C07311=1150.846,-117.168,-42.980,178.656,5.934,149.460
C07312=1150.851,-117.418,-42.971,178.654,5.933,149.460
C07313=1150.857,-117.668,-42.963,178.652,5.933,149.461
C07314=1150.862,-117.917,-42.954,178.650,5.933,149.461
C07315=1150.868,-118.167,-42.945,178.648,5.933,149.462
C07316=1150.873,-118.417,-42.936,178.646,5.932,149.462
C07317=1150.878,-118.667,-42.929,178.644,5.931,149.463
C07318=1150.883,-118.916,-42.920,178.642,5.931,149.463
C07319=1150.888,-119.166,-42.911,178.640,5.930,149.464
C07320=1150.894,-119.416,-42.903,178.638,5.931,149.464
C07321=1150.900,-119.666,-42.895,178.636,5.930,149.465
C07322=1150.905,-119.916,-42.886,178.634,5.930,149.465
C07323=1150.910,-120.165,-42.877,178.632,5.929,149.466
C07324=1150.915,-120.415,-42.868,178.630,5.929,149.466
C07325=1150.921,-120.665,-42.860,178.628,5.929,149.467
C07326=1150.926,-120.915,-42.851,178.627,5.929,149.467
C07327=1150.932,-121.165,-42.842,178.624,5.928,149.468
C07328=1150.937,-121.414,-42.834,178.622,5.928,149.469
C07329=1150.943,-121.664,-42.826,178.620,5.928,149.469
C07330=1150.948,-121.914,-42.817,178.619,5.928,149.470
C07331=1150.954,-122.163,-42.808,178.616,5.927,149.470
C07332=1150.959,-122.413,-42.801,178.615,5.927,149.471
C07333=1150.964,-122.663,-42.792,178.613,5.926,149.471
C07334=1150.969,-122.913,-42.783,178.611,5.926,149.472
C07335=1150.975,-123.163,-42.775,178.609,5.926,149.472
C07336=1150.980,-123.413,-42.766,178.606,5.925,149.473
C07337=1150.985,-123.663,-42.757,178.604,5.925,149.473
C07338=1150.991,-123.912,-42.749,178.602,5.924,149.474
C07339=1150.997,-124.162,-42.741,178.601,5.924,149.474
C07340=1151.001,-124.412,-42.733,178.598,5.924,149.475
C07341=1151.007,-124.662,-42.724,178.597,5.924,149.475
C07342=1151.012,-124.911,-42.716,178.595,5.923,149.476
C07343=1151.018,-125.162,-42.707,178.593,5.923,149.476
C07344=1151.023,-125.411,-42.699,178.591,5.922,149.477
C07345=1151.029,-125.661,-42.690,178.589,5.923,149.477
C07346=1151.034,-125.910,-42.683,178.587,5.922,149.478
C07347=1151.039,-126.160,-42.674,178.585,5.922,149.478
C07348=1151.045,-126.411,-42.666,178.583,5.921,149.479
C07349=1151.050,-126.660,-42.657,178.581,5.921,149.479
C07350=1151.056,-126.910,-42.649,178.579,5.921,149.480
C07351=1151.061,-127.160,-42.640,178.577,5.921,149.480
C07352=1151.066,-127.409,-42.632,178.575,5.920,149.481
C07353=1151.071,-127.659,-42.624,178.574,5.920,149.481
C07354=1151.077,-127.909,-42.615,178.571,5.919,149.482
C07355=1151.083,-128.159,-42.607,178.569,5.920,149.482
C07356=1150.661,-128.171,-42.650,178.566,5.922,149.484
C07357=1150.656,-127.920,-42.658,178.568,5.923,149.484
C07358=1150.651,-127.670,-42.667,178.570,5.923,149.483
C07359=1150.645,-127.420,-42.675,178.572,5.924,149.483
C07360=1150.640,-127.171,-42.683,178.574,5.924,149.482
C07361=1150.635,-126.922,-42.691,178.576,5.925,149.482
C07362=1150.629,-126.671,-42.700,178.577,5.925,149.481
C07363=1150.624,-126.421,-42.708,178.580,5.925,149.481
C07364=1150.618,-126.172,-42.716,178.581,5.925,149.480
C07365=1150.613,-125.922,-42.725,178.584,5.926,149.479
C07366=1150.608,-125.672,-42.733,178.585,5.926,149.479
C07367=1150.602,-125.423,-42.741,178.588,5.926,149.478
C07368=1150.597,-125.173,-42.750,178.589,5.926,149.478
C07369=1150.592,-124.922,-42.758,178.591,5.927,149.477
C07370=1150.586,-124.673,-42.767,178.593,5.927,149.477
C07371=1150.580,-124.423,-42.775,178.595,5.928,149.477
C07372=1150.576,-124.173,-42.783,178.597,5.928,149.476
C07373=1150.570,-123.924,-42.792,178.599,5.929,149.476
C07374=1150.565,-123.673,-42.800,178.601,5.928,149.475
C07375=1150.559,-123.424,-42.809,178.603,5.929,149.474
C07376=1150.554,-123.174,-42.818,178.605,5.929,149.474
C07377=1150.548,-122.924,-42.826,178.607,5.930,149.473
C07378=1150.543,-122.674,-42.835,178.609,5.929,149.473
C07379=1150.537,-122.425,-42.843,178.611,5.930,149.472
C07380=1150.533,-122.175,-42.851,178.612,5.930,149.472
C07381=1150.527,-121.925,-42.860,178.615,5.931,149.471
C07382=1150.522,-121.676,-42.868,178.617,5.932,149.471
C07383=1150.516,-121.425,-42.876,178.619,5.931,149.470
C07384=1150.511,-121.175,-42.885,178.621,5.932,149.470
C07385=1150.505,-120.926,-42.894,178.623,5.932,149.469
C07386=1150.500,-120.676,-42.902,178.625,5.933,149.469
C07387=1150.495,-120.426,-42.911,178.627,5.933,149.468
C07388=1150.489,-120.176,-42.920,178.629,5.933,149.468
C07389=1150.484,-119.927,-42.928,178.630,5.933,149.467
C07390=1150.478,-119.677,-42.936,178.633,5.934,149.467
C07391=1150.473,-119.427,-42.945,178.635,5.934,149.466
C07392=1150.467,-119.178,-42.954,178.637,5.934,149.466
C07393=1150.462,-118.928,-42.963,178.638,5.934,149.465
C07394=1150.457,-118.678,-42.970,178.641,5.935,149.465
C07395=1150.452,-118.428,-42.979,178.642,5.935,149.464
C07396=1150.446,-118.179,-42.988,178.644,5.936,149.464
C07397=1150.441,-117.929,-42.997,178.646,5.936,149.463
C07398=1150.436,-117.678,-43.005,178.649,5.936,149.462
C07399=1150.430,-117.429,-43.013,178.651,5.937,149.462
C07400=1150.425,-117.179,-43.022,178.652,5.937,149.461
C07401=1150.420,-116.929,-43.031,178.655,5.938,149.461
C07402=1150.415,-116.680,-43.040,178.656,5.938,149.460
C07403=1150.409,-116.430,-43.049,178.658,5.938,149.460
C07404=1150.403,-116.180,-43.057,178.660,5.938,149.460
C07405=1150.398,-115.930,-43.066,178.663,5.939,149.459
C07406=1150.393,-115.680,-43.075,178.664,5.939,149.458
C07407=1150.387,-115.431,-43.083,178.666,5.939,149.458
C07408=1150.382,-115.181,-43.092,178.668,5.939,149.457
C07409=1150.377,-114.931,-43.101,178.670,5.940,149.457
C07410=1150.371,-114.681,-43.110,178.672,5.941,149.456
C07411=1150.365,-114.431,-43.119,178.674,5.941,149.456
C07412=1150.360,-114.182,-43.127,178.677,5.941,149.455
C07413=1150.355,-113.932,-43.136,178.678,5.941,149.455
C07414=1150.349,-113.682,-43.145,178.681,5.942,149.454
C07415=1150.344,-113.432,-43.154,178.682,5.942,149.454
C07416=1150.338,-113.183,-43.162,178.684,5.943,149.453
C07417=1150.333,-112.933,-43.171,178.686,5.943,149.453
C07418=1150.328,-112.683,-43.180,178.689,5.943,149.452
C07419=1150.323,-112.433,-43.188,178.691,5.944,149.452
C07420=1150.317,-112.183,-43.197,178.692,5.944,149.451
C07421=1150.312,-111.934,-43.206,178.695,5.944,149.451
C07422=1150.307,-111.684,-43.215,178.696,5.944,149.450
C07423=1150.301,-111.434,-43.224,178.698,5.945,149.450
C07424=1150.295,-111.184,-43.233,178.700,5.945,149.449
C07425=1150.290,-110.934,-43.242,178.703,5.945,149.448
C07426=1150.285,-110.684,-43.251,178.705,5.946,149.448
C07427=1150.279,-110.435,-43.259,178.706,5.946,149.447
C07428=1150.274,-110.185,-43.268,178.709,5.947,149.447
C07429=1150.269,-109.935,-43.277,178.711,5.947,149.446
C07430=1150.264,-109.685,-43.286,178.713,5.947,149.446
C07431=1150.259,-109.436,-43.295,178.715,5.947,149.445
C07432=1150.254,-109.186,-43.304,178.717,5.948,149.445
C07433=1150.247,-108.936,-43.313,178.719,5.949,149.444
C07434=1150.242,-108.686,-43.322,178.721,5.949,149.444
C07435=1150.237,-108.437,-43.331,178.723,5.949,149.443
C07436=1150.232,-108.187,-43.340,178.725,5.949,149.443
C07437=1150.226,-107.937,-43.349,178.727,5.950,149.442
C07438=1150.221,-107.687,-43.358,178.729,5.950,149.442
C07439=1150.215,-107.437,-43.367,178.731,5.951,149.441
C07440=1150.210,-107.188,-43.376,178.733,5.951,149.440
C07441=1150.204,-106.938,-43.384,178.735,5.951,149.440
C07442=1150.199,-106.688,-43.393,178.737,5.952,149.439
C07443=1150.194,-106.438,-43.402,178.739,5.952,149.439
C07444=1150.189,-106.188,-43.411,178.741,5.952,149.438
C07445=1150.183,-105.939,-43.421,178.744,5.953,149.438
C07446=1150.178,-105.689,-43.430,178.745,5.953,149.437
C07447=1150.173,-105.439,-43.439,178.748,5.953,149.437
C07448=1150.168,-105.189,-43.448,178.749,5.953,149.436
C07449=1150.162,-104.940,-43.457,178.751,5.954,149.436
C07450=1150.156,-104.690,-43.466,178.753,5.954,149.435
C07451=1150.151,-104.440,-43.475,178.756,5.954,149.435
C07452=1150.146,-104.190,-43.484,178.758,5.955,149.434
C07453=1150.141,-103.941,-43.493,178.759,5.955,149.434
C07454=1150.135,-103.691,-43.503,178.762,5.956,149.433
C07455=1150.130,-103.441,-43.512,178.764,5.956,149.432
C07456=1150.125,-103.191,-43.521,178.766,5.956,149.432
C07457=1150.119,-102.919,-43.531,178.768,5.957,149.431
C07458=1150.113,-102.647,-43.540,178.771,5.957,149.431
C07459=1150.107,-102.375,-43.550,178.772,5.957,149.430
C07460=1150.101,-102.103,-43.560,178.775,5.958,149.430
C07461=1150.096,-101.853,-43.570,178.777,5.959,149.429
C07462=1150.091,-101.603,-43.579,178.779,5.958,149.429
C07463=1150.086,-101.354,-43.588,178.781,5.959,149.428
C07464=1150.080,-101.103,-43.597,178.784,5.960,149.427
C07465=1150.074,-100.854,-43.606,178.785,5.960,149.427
C07466=1150.070,-100.604,-43.616,178.787,5.960,149.426
C07467=1150.064,-100.354,-43.625,178.789,5.960,149.426
C07468=1150.059,-100.104,-43.634,178.791,5.961,149.425
C07469=1150.053,-99.854,-43.643,178.794,5.961,149.425
C07470=1150.049,-99.605,-43.653,178.795,5.961,149.424
C07471=1150.043,-99.355,-43.662,178.798,5.962,149.424
C07472=1150.037,-99.105,-43.671,178.799,5.962,149.423
C07473=1150.032,-98.855,-43.680,178.802,5.962,149.423
C07474=1150.027,-98.606,-43.690,178.804,5.963,149.422
C07475=1150.022,-98.356,-43.699,178.806,5.963,149.422
C07476=1150.016,-98.106,-43.709,178.808,5.964,149.421
C07477=1150.011,-97.857,-43.718,178.811,5.964,149.420
C07478=1150.006,-97.607,-43.727,178.812,5.964,149.420
C07479=1150.000,-97.357,-43.737,178.814,5.965,149.419
C07480=1149.995,-97.107,-43.746,178.816,5.965,149.419
C07481=1149.990,-96.857,-43.755,178.819,5.965,149.418
C07482=1149.984,-96.607,-43.765,178.821,5.966,149.418
C07483=1149.979,-96.358,-43.774,178.822,5.966,149.417
C07484=1149.974,-96.108,-43.783,178.825,5.967,149.417
C07485=1149.968,-95.858,-43.793,178.827,5.967,149.416
C07486=1149.963,-95.609,-43.802,178.829,5.967,149.416
C07487=1149.957,-95.359,-43.812,178.831,5.968,149.415
C07488=1149.952,-95.109,-43.821,178.833,5.968,149.415
C07489=1149.946,-94.859,-43.831,178.835,5.968,149.414
C07490=1149.941,-94.609,-43.840,178.838,5.969,149.413
C07491=1149.936,-94.360,-43.849,178.839,5.969,149.413
C07492=1149.930,-94.110,-43.859,178.841,5.970,149.412
C07493=1149.925,-93.860,-43.868,178.844,5.970,149.412
C07494=1149.920,-93.611,-43.878,178.846,5.970,149.411
C07495=1149.914,-93.361,-43.887,178.848,5.971,149.411
C07496=1149.909,-93.111,-43.897,178.850,5.972,149.410
C07497=1149.904,-92.861,-43.906,178.852,5.971,149.410
C07498=1149.898,-92.612,-43.915,178.854,5.972,149.409
C07499=1149.893,-92.362,-43.925,178.857,5.973,149.409
C07500=1149.888,-92.112,-43.934,178.858,5.973,149.408
C07501=1149.882,-91.863,-43.944,178.861,5.973,149.407
C07502=1149.877,-91.613,-43.953,178.863,5.974,149.407
C07503=1149.871,-91.363,-43.963,178.865,5.974,149.406
C07504=1149.867,-91.113,-43.973,178.867,5.975,149.406
C07505=1149.861,-90.863,-43.983,178.869,5.975,149.405
C07506=1149.856,-90.613,-43.992,178.871,5.975,149.405
C07507=1149.850,-90.364,-44.002,178.873,5.976,149.404
C07508=1149.845,-90.114,-44.011,178.875,5.975,149.404
C07509=1149.840,-89.864,-44.021,178.877,5.976,149.403
C07510=1149.834,-89.614,-44.030,178.880,5.977,149.403
C07511=1149.829,-89.365,-44.040,178.881,5.977,149.402
C07512=1149.824,-89.115,-44.049,178.884,5.977,149.401
C07513=1149.818,-88.866,-44.059,178.886,5.978,149.401
C07514=1149.814,-88.615,-44.068,178.888,5.978,149.400
C07515=1149.808,-88.365,-44.079,178.890,5.979,149.400
C07516=1149.803,-88.116,-44.088,178.893,5.979,149.399
C07517=1149.797,-87.866,-44.098,178.894,5.979,149.399
C07518=1149.792,-87.617,-44.107,178.896,5.980,149.398
C07519=1149.786,-87.367,-44.117,178.899,5.980,149.398
C07520=1149.781,-87.117,-44.127,178.901,5.981,149.397
C07521=1149.776,-86.867,-44.136,178.903,5.981,149.397
C07522=1149.771,-86.617,-44.147,178.905,5.982,149.396
C07523=1149.766,-86.368,-44.156,178.908,5.982,149.395
C07524=1149.760,-86.118,-44.166,178.909,5.982,149.395
C07525=1149.755,-85.868,-44.175,178.912,5.983,149.394
C07526=1149.749,-85.618,-44.185,178.914,5.983,149.394
C07527=1149.744,-85.369,-44.195,178.916,5.983,149.393
C07528=1149.739,-85.119,-44.205,178.918,5.984,149.393
C07529=1149.733,-84.869,-44.214,178.920,5.985,149.392
C07530=1149.729,-84.619,-44.224,178.922,5.984,149.392
C07531=1149.723,-84.370,-44.234,178.924,5.985,149.391
C07532=1149.717,-84.120,-44.244,178.927,5.986,149.391
C07533=1149.712,-83.870,-44.253,178.929,5.985,149.390
C07534=1149.707,-83.620,-44.264,178.931,5.986,149.389
C07535=1149.702,-83.370,-44.273,178.933,5.987,149.389
C07536=1149.696,-83.121,-44.283,178.935,5.987,149.388
C07537=1149.691,-82.871,-44.293,178.937,5.987,149.388
C07538=1149.686,-82.622,-44.303,178.940,5.988,149.387
C07539=1149.681,-82.371,-44.313,178.942,5.989,149.387
C07540=1149.675,-82.122,-44.323,178.944,5.988,149.386
C07541=1149.670,-81.872,-44.333,178.946,5.989,149.386
C07542=1149.665,-81.623,-44.343,178.948,5.990,149.385
C07543=1149.659,-81.373,-44.352,178.950,5.990,149.384
C07544=1149.654,-81.123,-44.362,178.952,5.990,149.384
C07545=1149.649,-80.873,-44.372,178.955,5.991,149.383
C07546=1149.643,-80.624,-44.383,178.957,5.991,149.383
C07547=1149.638,-80.374,-44.392,178.959,5.991,149.382
C07548=1149.633,-80.124,-44.402,178.961,5.992,149.382
C07549=1149.627,-79.874,-44.412,178.964,5.993,149.381
C07550=1149.622,-79.624,-44.423,178.965,5.993,149.381
C07551=1149.617,-79.375,-44.431,178.968,5.993,149.380
C07552=1149.611,-79.125,-44.442,178.970,5.994,149.379
C07553=1149.606,-78.875,-44.452,178.972,5.994,149.379
C07554=1149.601,-78.626,-44.462,178.974,5.994,149.378
C07555=1149.596,-78.376,-44.472,178.976,5.995,149.378
C07556=1149.590,-78.127,-44.482,178.979,5.996,149.377
C07557=1149.585,-77.876,-44.492,178.980,5.996,149.377
C07558=1149.580,-77.626,-44.502,178.983,5.996,149.376
C07559=1149.574,-77.377,-44.512,178.985,5.997,149.376
C07560=1149.569,-77.127,-44.522,178.988,5.997,149.375
C07561=1149.563,-76.856,-44.533,178.990,5.997,149.374
C07562=1149.558,-76.584,-44.545,178.992,5.998,149.374
C07563=1149.552,-76.312,-44.555,178.994,5.998,149.373
C07564=1149.546,-76.042,-44.566,178.997,5.999,149.373
C07565=1149.540,-75.792,-44.576,178.999,6.000,149.372
C07566=1149.536,-75.542,-44.586,179.001,5.999,149.371
C07567=1149.530,-75.293,-44.596,179.003,6.000,149.371
C07568=1149.524,-75.043,-44.607,179.005,6.001,149.370
C07569=1149.519,-74.793,-44.617,179.008,6.001,149.370
C07570=1149.514,-74.543,-44.627,179.010,6.001,149.369
C07571=1149.508,-74.294,-44.638,179.012,6.002,149.369
C07572=1149.504,-74.044,-44.648,179.014,6.002,149.368
C07573=1149.498,-73.794,-44.658,179.017,6.003,149.368
C07574=1149.493,-73.545,-44.668,179.018,6.003,149.367
C07575=1149.487,-73.295,-44.678,179.021,6.004,149.366
C07576=1149.482,-73.044,-44.688,179.023,6.004,149.366
C07577=1149.476,-72.795,-44.698,179.025,6.005,149.365
C07578=1149.471,-72.545,-44.708,179.027,6.005,149.365
C07579=1149.466,-72.295,-44.719,179.030,6.005,149.364
C07580=1149.461,-72.046,-44.729,179.032,6.006,149.364
C07581=1149.455,-71.796,-44.739,179.034,6.007,149.363
C07582=1149.451,-71.547,-44.750,179.036,6.007,149.363
C07583=1149.445,-71.297,-44.760,179.039,6.007,149.362
C07584=1149.439,-71.047,-44.771,179.041,6.008,149.361
C07585=1149.434,-70.797,-44.781,179.043,6.008,149.361
C07586=1149.429,-70.548,-44.791,179.045,6.008,149.360
C07587=1149.425,-70.298,-44.801,179.047,6.009,149.360
C07588=1149.419,-70.048,-44.812,179.050,6.010,149.359
C07589=1149.413,-69.799,-44.822,179.052,6.010,149.359
C07590=1149.408,-69.548,-44.832,179.054,6.010,149.358
C07591=1149.403,-69.299,-44.843,179.056,6.011,149.358
C07592=1149.397,-69.049,-44.853,179.059,6.011,149.357
C07593=1149.392,-68.799,-44.863,179.061,6.012,149.356
C07594=1149.387,-68.550,-44.874,179.062,6.012,149.356
C07595=1149.382,-68.299,-44.884,179.065,6.012,149.355
C07596=1149.376,-68.050,-44.895,179.067,6.013,149.355
C07597=1149.371,-67.801,-44.905,179.069,6.014,149.354
C07598=1149.366,-67.551,-44.916,179.072,6.014,149.354
C07599=1149.360,-67.301,-44.926,179.074,6.014,149.353
C07600=1149.355,-67.051,-44.937,179.076,6.015,149.353
C07601=1149.349,-66.801,-44.947,179.079,6.015,149.352
C07602=1149.344,-66.552,-44.957,179.081,6.016,149.351
C07603=1149.339,-66.302,-44.968,179.083,6.016,149.351
C07604=1149.334,-66.053,-44.979,179.085,6.017,149.350
C07605=1149.329,-65.802,-44.989,179.087,6.017,149.350
C07606=1149.323,-65.553,-44.999,179.090,6.018,149.349
C07607=1149.318,-65.302,-45.010,179.092,6.018,149.349
C07608=1149.313,-65.054,-45.021,179.094,6.018,149.348
C07609=1149.307,-64.804,-45.031,179.096,6.019,149.347
C07610=1149.302,-64.554,-45.042,179.099,6.020,149.347
C07611=1149.297,-64.304,-45.052,179.101,6.020,149.346
C07612=1149.292,-64.055,-45.063,179.103,6.021,149.346
C07613=1149.286,-63.805,-45.073,179.105,6.021,149.345
C07614=1149.281,-63.555,-45.084,179.107,6.022,149.345
C07615=1149.276,-63.305,-45.094,179.110,6.022,149.344
C07616=1149.271,-63.056,-45.105,179.112,6.023,149.344
C07617=1149.265,-62.806,-45.116,179.114,6.022,149.343
C07618=1149.260,-62.556,-45.126,179.116,6.023,149.342
C07619=1149.255,-62.306,-45.136,179.119,6.024,149.342
C07620=1149.250,-62.057,-45.148,179.121,6.024,149.341
C07621=1149.244,-61.807,-45.158,179.123,6.025,149.341
C07622=1149.239,-61.558,-45.168,179.125,6.025,149.340
C07623=1149.234,-61.308,-45.179,179.128,6.025,149.340
C07624=1149.229,-61.058,-45.190,179.130,6.026,149.339
C07625=1149.224,-60.808,-45.200,179.132,6.027,149.338
C07626=1149.218,-60.559,-45.212,179.135,6.027,149.338
C07627=1149.213,-60.309,-45.222,179.137,6.028,149.337
C07628=1149.208,-60.058,-45.233,179.139,6.028,149.337
C07629=1149.202,-59.810,-45.244,179.141,6.029,149.336
C07630=1149.197,-59.559,-45.254,179.143,6.029,149.336
C07631=1149.192,-59.310,-45.265,179.146,6.030,149.335
C07632=1149.187,-59.060,-45.276,179.148,6.030,149.335
C07633=1149.181,-58.811,-45.286,179.150,6.030,149.334
C07634=1149.177,-58.561,-45.297,179.152,6.031,149.333
C07635=1149.170,-58.311,-45.308,179.155,6.032,149.333
C07636=1149.166,-58.061,-45.319,179.157,6.032,149.332
C07637=1149.160,-57.812,-45.330,179.159,6.033,149.332
C07638=1149.155,-57.562,-45.340,179.162,6.034,149.331
C07639=1149.150,-57.313,-45.351,179.164,6.033,149.331
C07640=1149.145,-57.063,-45.362,179.166,6.034,149.330
C07641=1149.139,-56.813,-45.374,179.169,6.034,149.329
C07642=1149.134,-56.563,-45.384,179.171,6.035,149.329
C07643=1149.129,-56.313,-45.395,179.173,6.036,149.328
C07644=1149.123,-56.064,-45.405,179.176,6.036,149.328
C07645=1149.119,-55.814,-45.417,179.177,6.036,149.327
C07646=1149.113,-55.565,-45.427,179.180,6.037,149.326
C07647=1149.108,-55.315,-45.439,179.182,6.037,149.326
C07648=1149.103,-55.065,-45.449,179.184,6.038,149.326
C07649=1149.097,-54.816,-45.460,179.187,6.039,149.325
C07650=1149.092,-54.565,-45.471,179.189,6.039,149.324
C07651=1149.086,-54.316,-45.482,179.191,6.039,149.324
C07652=1149.081,-54.066,-45.493,179.193,6.040,149.323
C07653=1149.077,-53.816,-45.504,179.196,6.041,149.323
C07654=1149.071,-53.567,-45.514,179.198,6.041,149.322
C07655=1149.066,-53.317,-45.526,179.200,6.042,149.321
C07656=1149.060,-53.067,-45.536,179.203,6.043,149.321
C07657=1149.055,-52.818,-45.548,179.205,6.042,149.320
C07658=1149.051,-52.568,-45.559,179.207,6.043,149.320
C07659=1149.044,-52.318,-45.570,179.210,6.043,149.319
C07660=1149.040,-52.068,-45.581,179.212,6.044,149.319
C07661=1149.034,-51.819,-45.591,179.214,6.045,149.318
C07662=1149.029,-51.569,-45.603,179.217,6.045,149.317
C07663=1149.024,-51.319,-45.615,179.219,6.046,149.317
C07664=1149.018,-51.070,-45.625,179.221,6.046,149.316
C07665=1149.013,-50.799,-45.637,179.223,6.046,149.316
C07666=1149.007,-50.528,-45.649,179.226,6.047,149.315
C07667=1149.002,-50.258,-45.661,179.228,6.048,149.315
C07668=1148.996,-49.987,-45.673,179.231,6.049,149.314
C07669=1148.991,-49.737,-45.685,179.233,6.049,149.313
C07670=1148.985,-49.488,-45.696,179.235,6.049,149.313
C07671=1148.980,-49.238,-45.706,179.238,6.050,149.312
C07672=1148.975,-48.988,-45.718,179.240,6.050,149.312
C07673=1148.970,-48.739,-45.729,179.242,6.051,149.311
C07674=1148.965,-48.489,-45.740,179.245,6.052,149.311
C07675=1148.959,-48.239,-45.751,179.247,6.052,149.310
C07676=1148.954,-47.990,-45.762,179.249,6.052,149.309
C07677=1148.948,-47.740,-45.774,179.252,6.053,149.309
C07678=1148.943,-47.490,-45.785,179.254,6.054,149.308
C07679=1148.938,-47.241,-45.796,179.256,6.054,149.308
C07680=1148.933,-46.991,-45.808,179.259,6.055,149.307
C07681=1148.928,-46.741,-45.819,179.261,6.056,149.307
C07682=1148.922,-46.491,-45.830,179.263,6.056,149.306
C07683=1148.917,-46.242,-45.841,179.266,6.057,149.305
C07684=1148.912,-45.992,-45.852,179.268,6.057,149.305
C07685=1148.907,-45.742,-45.864,179.270,6.057,149.304
C07686=1148.901,-45.493,-45.874,179.272,6.058,149.304
C07687=1148.896,-45.243,-45.886,179.275,6.058,149.303
C07688=1148.891,-44.993,-45.898,179.277,6.059,149.303
C07689=1148.885,-44.744,-45.909,179.280,6.059,149.302
C07690=1148.880,-44.494,-45.920,179.282,6.060,149.301
C07691=1148.875,-44.244,-45.931,179.284,6.061,149.301
C07692=1148.870,-43.994,-45.943,179.287,6.061,149.300
C07693=1148.865,-43.745,-45.954,179.289,6.062,149.300
C07694=1148.859,-43.495,-45.966,179.291,6.062,149.299
C07695=1148.855,-43.246,-45.977,179.293,6.063,149.299
C07696=1148.849,-42.996,-45.989,179.295,6.063,149.298
C07697=1148.844,-42.747,-46.000,179.298,6.064,149.297
C07698=1148.838,-42.497,-46.012,179.300,6.065,149.297
C07699=1148.833,-42.246,-46.022,179.303,6.065,149.296
C07700=1148.828,-41.997,-46.034,179.305,6.066,149.296
C07701=1148.823,-41.747,-46.045,179.307,6.067,149.295
C07702=1148.817,-41.498,-46.057,179.310,6.067,149.295
C07703=1148.813,-41.248,-46.068,179.312,6.068,149.294
C07704=1148.807,-40.998,-46.080,179.315,6.068,149.293
C07705=1148.802,-40.749,-46.091,179.317,6.069,149.293
C07706=1148.796,-40.499,-46.103,179.319,6.069,149.292
C07707=1148.792,-40.250,-46.114,179.321,6.069,149.292
C07708=1148.786,-40.000,-46.126,179.323,6.070,149.291
C07709=1148.781,-39.750,-46.138,179.326,6.071,149.291
C07710=1148.776,-39.500,-46.149,179.328,6.071,149.290
C07711=1148.770,-39.251,-46.161,179.331,6.072,149.289
C07712=1148.765,-39.001,-46.172,179.333,6.073,149.289
C07713=1148.760,-38.751,-46.184,179.335,6.073,149.288
C07714=1148.755,-38.502,-46.195,179.338,6.074,149.288
C07715=1148.750,-38.252,-46.207,179.340,6.075,149.287
C07716=1148.744,-38.002,-46.219,179.343,6.075,149.287
C07717=1148.739,-37.753,-46.230,179.345,6.076,149.286
C07718=1148.734,-37.503,-46.242,179.348,6.076,149.285
C07719=1148.729,-37.253,-46.253,179.349,6.076,149.285
C07720=1148.724,-37.003,-46.265,179.351,6.077,149.284
C07721=1148.718,-36.753,-46.277,179.354,6.077,149.284
C07722=1148.714,-36.504,-46.288,179.356,6.078,149.283
C07723=1148.707,-36.255,-46.300,179.359,6.079,149.283
C07724=1148.702,-36.005,-46.312,179.361,6.079,149.282
C07725=1148.697,-35.755,-46.323,179.364,6.080,149.281
C07726=1148.692,-35.505,-46.335,179.366,6.081,149.281
C07727=1148.688,-35.256,-46.347,179.368,6.081,149.280
C07728=1148.682,-35.006,-46.359,179.371,6.082,149.280
C07729=1148.677,-34.756,-46.370,179.373,6.083,149.279
C07730=1148.672,-34.507,-46.382,179.376,6.083,149.279
C07731=1148.666,-34.257,-46.393,179.378,6.084,149.278
C07732=1148.661,-34.007,-46.405,179.380,6.084,149.277
C07733=1148.655,-33.758,-46.417,179.383,6.085,149.277
C07734=1148.651,-33.509,-46.429,179.385,6.086,149.276
C07735=1148.645,-33.259,-46.441,179.387,6.086,149.276
C07736=1148.640,-33.009,-46.453,179.390,6.087,149.275
C07737=1148.635,-32.759,-46.464,179.392,6.087,149.275
C07738=1148.630,-32.509,-46.476,179.395,6.088,149.274
C07739=1148.624,-32.259,-46.488,179.397,6.089,149.273
C07740=1148.620,-32.010,-46.500,179.399,6.089,149.273
C07741=1148.614,-31.761,-46.511,179.401,6.089,149.272
C07742=1148.608,-31.511,-46.523,179.404,6.090,149.272
C07743=1148.603,-31.261,-46.535,179.406,6.091,149.271
C07744=1148.599,-31.012,-46.547,179.408,6.091,149.271
C07745=1148.593,-30.762,-46.559,179.411,6.092,149.270
C07746=1148.588,-30.512,-46.571,179.413,6.092,149.269
C07747=1148.582,-30.262,-46.583,179.415,6.093,149.269
C07748=1148.578,-30.013,-46.595,179.418,6.094,149.268
C07749=1148.573,-29.763,-46.607,179.420,6.094,149.268
C07750=1148.567,-29.513,-46.619,179.422,6.095,149.267
C07751=1148.562,-29.264,-46.631,179.425,6.095,149.267
C07752=1148.557,-29.014,-46.643,179.427,6.096,149.266
C07753=1148.552,-28.764,-46.654,179.430,6.097,149.265
C07754=1148.546,-28.515,-46.666,179.432,6.097,149.265
C07755=1148.541,-28.265,-46.679,179.434,6.098,149.264
C07756=1148.536,-28.015,-46.691,179.437,6.099,149.264
C07757=1148.530,-27.765,-46.703,179.439,6.099,149.263
C07758=1148.526,-27.516,-46.715,179.442,6.100,149.263
C07759=1148.521,-27.266,-46.727,179.444,6.101,149.262
C07760=1148.516,-27.017,-46.739,179.447,6.101,149.261
C07761=1148.510,-26.767,-46.751,179.449,6.102,149.261
C07762=1148.505,-26.517,-46.763,179.452,6.102,149.260
C07763=1148.500,-26.268,-46.776,179.454,6.103,149.260
C07764=1148.495,-26.018,-46.787,179.456,6.104,149.259
C07765=1148.490,-25.769,-46.799,179.459,6.104,149.259
C07766=1148.484,-25.519,-46.811,179.461,6.105,149.258
C07767=1148.479,-25.269,-46.823,179.463,6.105,149.257
C07768=1148.474,-25.020,-46.836,179.466,6.106,149.257
C07769=1148.468,-24.749,-46.849,179.468,6.107,149.256
C07770=1148.463,-24.480,-46.861,179.470,6.107,149.256
C07771=1148.457,-24.210,-46.876,179.474,6.109,149.255
C07772=1148.451,-23.939,-46.889,179.476,6.109,149.254
C07773=1148.446,-23.689,-46.900,179.479,6.110,149.254
C07774=1148.441,-23.440,-46.913,179.481,6.110,149.253
C07775=1148.435,-23.190,-46.925,179.483,6.111,149.253
C07776=1148.430,-22.941,-46.938,179.486,6.112,149.252
C07777=1148.425,-22.691,-46.949,179.488,6.112,149.252
C07778=1148.421,-22.442,-46.961,179.490,6.113,149.251
C07779=1148.415,-22.192,-46.973,179.493,6.114,149.250
C07780=1148.410,-21.943,-46.986,179.495,6.114,149.250
C07781=1148.405,-21.693,-46.999,179.498,6.115,149.249
C07782=1148.399,-21.443,-47.010,179.500,6.116,149.249
C07783=1148.394,-21.194,-47.023,179.503,6.116,149.248
C07784=1148.389,-20.944,-47.035,179.505,6.117,149.248
C07785=1148.384,-20.695,-47.048,179.507,6.118,149.247
C07786=1148.378,-20.445,-47.059,179.510,6.118,149.246
C07787=1148.374,-20.195,-47.072,179.512,6.119,149.246
C07788=1148.369,-19.946,-47.085,179.515,6.119,149.245
C07789=1148.363,-19.696,-47.097,179.517,6.120,149.245
C07790=1148.358,-19.446,-47.109,179.520,6.120,149.244
C07791=1148.353,-19.196,-47.121,179.522,6.121,149.244
C07792=1148.348,-18.947,-47.134,179.524,6.122,149.243
C07793=1148.342,-18.698,-47.147,179.527,6.122,149.243
C07794=1148.337,-18.448,-47.158,179.529,6.123,149.242
C07795=1148.333,-18.198,-47.171,179.532,6.124,149.241
C07796=1148.327,-17.948,-47.185,179.534,6.125,149.241
C07797=1148.321,-17.698,-47.196,179.537,6.126,149.240
C07798=1148.316,-17.449,-47.209,179.539,6.126,149.240
C07799=1148.311,-17.200,-47.222,179.542,6.127,149.239
C07800=1148.306,-16.950,-47.234,179.544,6.128,149.239
C07801=1148.300,-16.700,-47.246,179.546,6.128,149.238
C07802=1148.296,-16.450,-47.259,179.549,6.129,149.237
C07803=1148.290,-16.200,-47.271,179.551,6.130,149.237
C07804=1148.285,-15.951,-47.284,179.554,6.130,149.236
C07805=1148.280,-15.702,-47.296,179.556,6.131,149.236
C07806=1148.275,-15.452,-47.309,179.558,6.131,149.235
C07807=1148.270,-15.202,-47.321,179.561,6.132,149.235
C07808=1148.264,-14.952,-47.334,179.563,6.133,149.234
C07809=1148.259,-14.703,-47.347,179.565,6.133,149.233
C07810=1148.254,-14.453,-47.359,179.568,6.134,149.233
C07811=1148.249,-14.204,-47.372,179.570,6.135,149.232
C07812=1148.244,-13.954,-47.384,179.573,6.136,149.232
C07813=1148.239,-13.704,-47.397,179.576,6.137,149.231
C07814=1148.234,-13.455,-47.410,179.578,6.137,149.231
C07815=1148.228,-13.205,-47.423,179.580,6.138,149.230
C07816=1148.223,-12.956,-47.435,179.583,6.139,149.229
C07817=1148.218,-12.706,-47.447,179.585,6.139,149.229
C07818=1148.213,-12.456,-47.460,179.587,6.140,149.228
C07819=1148.208,-12.207,-47.473,179.590,6.140,149.228
C07820=1148.203,-11.957,-47.485,179.592,6.141,149.227
C07821=1148.197,-11.708,-47.499,179.595,6.142,149.226
C07822=1148.192,-11.458,-47.512,179.597,6.142,149.226
C07823=1148.187,-11.208,-47.524,179.599,6.143,149.226
C07824=1148.182,-10.959,-47.537,179.603,6.144,149.225
C07825=1148.177,-10.709,-47.549,179.605,6.145,149.224
C07826=1148.171,-10.459,-47.562,179.607,6.146,149.224
C07827=1148.166,-10.209,-47.575,179.610,6.146,149.223
C07828=1148.161,-9.960,-47.587,179.612,6.147,149.223
C07829=1148.156,-9.711,-47.600,179.614,6.148,149.222
C07830=1148.151,-9.461,-47.614,179.617,6.148,149.221
C07831=1148.146,-9.211,-47.626,179.619,6.149,149.221
C07832=1148.141,-8.962,-47.639,179.621,6.150,149.220
C07833=1148.136,-8.712,-47.652,179.624,6.150,149.220
C07834=1148.130,-8.462,-47.665,179.627,6.152,149.219
C07835=1148.125,-8.213,-47.678,179.630,6.152,149.219
C07836=1148.120,-7.964,-47.690,179.632,6.153,149.218
C07837=1148.115,-7.714,-47.703,179.634,6.153,149.217
C07838=1148.110,-7.464,-47.716,179.637,6.154,149.217
C07839=1148.104,-7.215,-47.729,179.639,6.155,149.216
C07840=1148.100,-6.965,-47.742,179.641,6.155,149.216
C07841=1148.094,-6.715,-47.755,179.644,6.156,149.215
C07842=1148.089,-6.466,-47.768,179.646,6.157,149.215
C07843=1148.084,-6.216,-47.781,179.649,6.158,149.214
C07844=1148.079,-5.966,-47.794,179.652,6.159,149.213
C07845=1148.073,-5.717,-47.806,179.654,6.160,149.213
C07846=1148.069,-5.467,-47.819,179.657,6.160,149.212
C07847=1148.063,-5.218,-47.833,179.659,6.161,149.212
C07848=1148.058,-4.968,-47.846,179.661,6.161,149.211
C07849=1148.054,-4.718,-47.859,179.664,6.162,149.211
C07850=1148.048,-4.469,-47.872,179.666,6.162,149.210
C07851=1148.043,-4.219,-47.885,179.669,6.164,149.210
C07852=1148.038,-3.969,-47.898,179.671,6.165,149.209
C07853=1148.032,-3.720,-47.911,179.674,6.165,149.208
C07854=1148.027,-3.470,-47.923,179.676,6.166,149.208
C07855=1148.022,-3.221,-47.938,179.679,6.167,149.207
C07856=1148.017,-2.971,-47.950,179.681,6.167,149.207
C07857=1148.013,-2.721,-47.963,179.683,6.168,149.206
C07858=1148.007,-2.472,-47.976,179.686,6.169,149.206
C07859=1148.002,-2.222,-47.989,179.689,6.170,149.205
C07860=1147.996,-1.972,-48.003,179.691,6.171,149.204
C07861=1147.992,-1.723,-48.016,179.693,6.171,149.204
C07862=1147.987,-1.473,-48.029,179.696,6.172,149.203
C07863=1147.981,-1.224,-48.042,179.698,6.173,149.203
C07864=1147.976,-0.974,-48.055,179.701,6.173,149.202
C07865=1147.971,-0.725,-48.069,179.703,6.175,149.202
C07866=1147.966,-0.475,-48.082,179.706,6.175,149.201
C07867=1147.961,-0.225,-48.095,179.708,6.176,149.201
C07868=1147.956,0.024,-48.108,179.711,6.176,149.200
C07869=1147.950,0.273,-48.122,179.713,6.177,149.199
C07870=1147.945,0.523,-48.135,179.716,6.178,149.199
C07871=1147.940,0.773,-48.148,179.719,6.179,149.198
C07872=1147.935,1.023,-48.161,179.721,6.180,149.198
C07873=1147.929,1.292,-48.175,179.723,6.181,149.197
C07874=1147.923,1.562,-48.190,179.726,6.181,149.196
C07875=1147.919,1.831,-48.204,179.729,6.183,149.196
C07876=1147.913,2.101,-48.218,179.731,6.183,149.195
C07877=1147.907,2.350,-48.232,179.734,6.184,149.195
C07878=1147.903,2.600,-48.245,179.736,6.184,149.194
C07879=1147.897,2.849,-48.259,179.739,6.186,149.194
C07880=1147.892,3.098,-48.272,179.742,6.186,149.193
C07881=1147.887,3.348,-48.285,179.744,6.187,149.192
C07882=1147.882,3.597,-48.299,179.747,6.188,149.192
C07883=1147.877,3.848,-48.312,179.749,6.188,149.191
C07884=1147.872,4.096,-48.325,179.752,6.190,149.191
C07885=1147.867,4.347,-48.339,179.754,6.190,149.190
C07886=1147.861,4.596,-48.352,179.756,6.191,149.190
C07887=1147.857,4.846,-48.366,179.759,6.192,149.189
C07888=1147.851,5.095,-48.379,179.761,6.193,149.189
C07889=1147.847,5.345,-48.393,179.764,6.193,149.188
C07890=1147.841,5.594,-48.406,179.767,6.195,149.187
C07891=1147.836,5.844,-48.420,179.769,6.195,149.187
C07892=1147.831,6.094,-48.433,179.771,6.196,149.186
C07893=1147.826,6.343,-48.447,179.774,6.196,149.186
C07894=1147.821,6.593,-48.460,179.776,6.197,149.185
C07895=1147.816,6.842,-48.474,179.779,6.199,149.185
C07896=1147.810,7.092,-48.488,179.782,6.199,149.184
C07897=1147.806,7.341,-48.501,179.784,6.200,149.183
C07898=1147.800,7.591,-48.514,179.787,6.200,149.183
C07899=1147.795,7.840,-48.528,179.789,6.202,149.182
C07900=1147.790,8.090,-48.541,179.792,6.202,149.182
C07901=1147.785,8.339,-48.555,179.794,6.203,149.181
C07902=1147.779,8.590,-48.569,179.797,6.204,149.181
C07903=1147.775,8.839,-48.583,179.799,6.205,149.180
C07904=1147.769,9.089,-48.596,179.802,6.206,149.180
C07905=1147.764,9.338,-48.610,179.804,6.207,149.179
C07906=1147.759,9.587,-48.624,179.807,6.207,149.178
C07907=1147.754,9.837,-48.637,179.809,6.208,149.178
C07908=1147.749,10.086,-48.651,179.811,6.209,149.177
C07909=1147.744,10.336,-48.665,179.815,6.210,149.177
C07910=1147.739,10.586,-48.678,179.817,6.211,149.176
C07911=1147.734,10.835,-48.692,179.819,6.211,149.175
C07912=1147.728,11.086,-48.705,179.822,6.212,149.175
C07913=1147.723,11.335,-48.719,179.824,6.214,149.175
C07914=1147.719,11.584,-48.733,179.827,6.214,149.174
C07915=1147.713,11.834,-48.747,179.829,6.215,149.173
C07916=1147.708,12.083,-48.761,179.832,6.215,149.173
C07917=1147.703,12.333,-48.775,179.835,6.217,149.172
C07918=1147.698,12.583,-48.789,179.837,6.217,149.172
C07919=1147.693,12.832,-48.802,179.839,6.218,149.171
C07920=1147.688,13.082,-48.816,179.842,6.219,149.170
C07921=1147.682,13.331,-48.830,179.844,6.219,149.170
C07922=1147.677,13.581,-48.843,179.847,6.221,149.170
C07923=1147.672,13.831,-48.858,179.850,6.222,149.169
C07924=1147.667,14.079,-48.871,179.852,6.222,149.168
C07925=1147.662,14.329,-48.885,179.854,6.223,149.168
C07926=1147.657,14.580,-48.899,179.857,6.224,149.167
C07927=1147.651,14.829,-48.913,179.860,6.225,149.167
C07928=1147.646,15.078,-48.927,179.862,6.226,149.166
C07929=1147.642,15.328,-48.941,179.865,6.227,149.165
C07930=1147.637,15.577,-48.955,179.868,6.228,149.165
C07931=1147.631,15.827,-48.968,179.870,6.229,149.164
C07932=1147.627,16.077,-48.983,179.872,6.229,149.164
C07933=1147.622,16.326,-48.997,179.875,6.231,149.163
C07934=1147.616,16.575,-49.011,179.878,6.231,149.163
C07935=1147.611,16.825,-49.025,179.880,6.232,149.162
C07936=1147.606,17.075,-49.039,179.883,6.232,149.162
C07937=1147.601,17.324,-49.053,179.885,6.234,149.161
C07938=1147.596,17.574,-49.066,179.887,6.235,149.161
C07939=1147.591,17.824,-49.080,179.890,6.235,149.160
C07940=1147.585,18.073,-49.094,179.892,6.236,149.159
C07941=1147.581,18.322,-49.109,179.896,6.237,149.159
C07942=1147.576,18.572,-49.123,179.898,6.238,149.158
C07943=1147.571,18.822,-49.137,179.900,6.239,149.158
C07944=1147.565,19.071,-49.151,179.903,6.240,149.157
C07945=1147.560,19.320,-49.165,179.906,6.241,149.156
C07946=1147.555,19.570,-49.180,179.908,6.242,149.156
C07947=1147.550,19.820,-49.194,179.910,6.242,149.156
C07948=1147.545,20.069,-49.208,179.913,6.244,149.155
C07949=1147.540,20.319,-49.222,179.916,6.244,149.154
C07950=1147.535,20.568,-49.236,179.918,6.245,149.154
C07951=1147.530,20.818,-49.251,179.921,6.246,149.153
C07952=1147.524,21.067,-49.265,179.924,6.247,149.153
C07953=1147.519,21.317,-49.279,179.926,6.248,149.152
C07954=1147.514,21.566,-49.293,179.928,6.249,149.152
C07955=1147.509,21.816,-49.307,179.931,6.250,149.151
C07956=1147.504,22.066,-49.322,179.933,6.251,149.151
C07957=1147.499,22.315,-49.336,179.936,6.251,149.150
C07958=1147.494,22.565,-49.350,179.939,6.253,149.149
C07959=1147.489,22.814,-49.364,179.941,6.253,149.149
C07960=1147.484,23.064,-49.378,179.944,6.254,149.148
C07961=1147.479,23.314,-49.393,179.946,6.256,149.148
C07962=1147.473,23.563,-49.407,179.949,6.256,149.147
C07963=1147.469,23.812,-49.421,179.951,6.257,149.147
C07964=1147.464,24.062,-49.435,179.954,6.258,149.146
C07965=1147.459,24.311,-49.450,179.957,6.259,149.146
C07966=1147.454,24.561,-49.464,179.959,6.259,149.145
C07967=1147.449,24.811,-49.479,179.961,6.260,149.144
C07968=1147.443,25.060,-49.493,179.964,6.262,149.144
C07969=1147.438,25.310,-49.507,179.967,6.262,149.143
C07970=1147.433,25.559,-49.522,179.969,6.263,149.143
C07971=1147.428,25.808,-49.537,179.972,6.264,149.142
C07972=1147.423,26.058,-49.551,179.974,6.265,149.142
C07973=1147.418,26.308,-49.565,179.977,6.266,149.141
C07974=1147.413,26.557,-49.579,179.980,6.267,149.141
C07975=1147.408,26.807,-49.593,179.982,6.268,149.140
C07976=1147.403,27.056,-49.608,179.985,6.269,149.139
C07977=1147.397,27.325,-49.624,179.987,6.270,149.139
C07978=1147.392,27.594,-49.640,179.990,6.271,149.138
C07979=1147.387,27.863,-49.655,179.993,6.272,149.138
C07980=1147.381,28.132,-49.672,179.995,6.273,149.137
C07981=1147.376,28.382,-49.686,179.999,6.274,149.137
C07982=1147.371,28.632,-49.700,-179.999,6.275,149.136
C07983=1147.366,28.881,-49.715,-179.996,6.276,149.135
C07984=1147.361,29.130,-49.729,-179.994,6.277,149.135
C07985=1147.356,29.379,-49.744,-179.992,6.278,149.134
C07986=1147.350,29.629,-49.758,-179.988,6.279,149.134
C07987=1147.345,29.878,-49.773,-179.986,6.280,149.133
C07988=1147.340,30.128,-49.788,-179.984,6.280,149.133
C07989=1147.335,30.378,-49.802,-179.981,6.282,149.132
C07990=1147.330,30.627,-49.818,-179.978,6.282,149.132
C07991=1147.325,30.877,-49.832,-179.976,6.283,149.131
C07992=1147.320,31.127,-49.846,-179.973,6.285,149.131
C07993=1147.316,31.376,-49.861,-179.971,6.285,149.130
C07994=1147.310,31.626,-49.876,-179.968,6.286,149.130
C07995=1147.305,31.875,-49.891,-179.965,6.287,149.129
C07996=1147.300,32.125,-49.905,-179.963,6.288,149.128
C07997=1147.295,32.374,-49.919,-179.960,6.290,149.128
C07998=1147.290,32.624,-49.935,-179.958,6.290,149.127
C07999=1147.285,32.873,-49.949,-179.955,6.291,149.127
C08000=1147.280,33.123,-49.964,-179.952,6.293,149.126
C08001=1147.275,33.373,-49.979,-179.950,6.293,149.126
C08002=1147.270,33.622,-49.994,-179.947,6.294,149.125
C08003=1147.264,33.871,-50.008,-179.945,6.295,149.125
C08004=1147.259,34.120,-50.024,-179.942,6.296,149.124
C08005=1147.254,34.370,-50.038,-179.939,6.298,149.123
C08006=1147.249,34.619,-50.053,-179.937,6.298,149.123
C08007=1147.244,34.869,-50.068,-179.934,6.299,149.122
C08008=1147.240,35.119,-50.083,-179.932,6.300,149.122
C08009=1147.235,35.368,-50.097,-179.929,6.301,149.121
C08010=1147.229,35.618,-50.113,-179.927,6.302,149.121
C08011=1147.224,35.868,-50.127,-179.924,6.303,149.120
C08012=1147.220,36.117,-50.142,-179.921,6.304,149.120
C08013=1147.214,36.367,-50.157,-179.919,6.306,149.119
C08014=1147.209,36.616,-50.172,-179.916,6.306,149.119
C08015=1147.204,36.866,-50.187,-179.914,6.307,149.118
C08016=1147.199,37.115,-50.202,-179.911,6.308,149.118
C08017=1147.194,37.364,-50.217,-179.908,6.309,149.117
C08018=1147.189,37.614,-50.232,-179.906,6.311,149.116
C08019=1147.184,37.863,-50.247,-179.904,6.311,149.116
C08020=1147.179,38.112,-50.263,-179.900,6.313,149.115
C08021=1147.174,38.362,-50.277,-179.898,6.313,149.115
C08022=1147.168,38.612,-50.292,-179.895,6.314,149.114
C08023=1147.163,38.861,-50.307,-179.893,6.316,149.114
C08024=1147.158,39.111,-50.322,-179.890,6.316,149.113
C08025=1147.153,39.360,-50.337,-179.887,6.318,149.113
C08026=1147.148,39.609,-50.353,-179.885,6.319,149.112
C08027=1147.143,39.859,-50.367,-179.883,6.319,149.111
C08028=1147.138,40.109,-50.383,-179.880,6.321,149.111
C08029=1147.134,40.358,-50.398,-179.877,6.321,149.110
C08030=1147.128,40.608,-50.413,-179.874,6.323,149.110
C08031=1147.123,40.857,-50.428,-179.872,6.324,149.109
C08032=1147.118,41.107,-50.444,-179.869,6.325,149.109
C08033=1147.113,41.356,-50.459,-179.867,6.326,149.108
C08034=1147.107,41.606,-50.473,-179.864,6.326,149.108
C08035=1147.103,41.855,-50.488,-179.861,6.328,149.107
C08036=1147.097,42.104,-50.504,-179.859,6.329,149.107
C08037=1147.093,42.354,-50.519,-179.856,6.330,149.106
C08038=1147.088,42.604,-50.534,-179.854,6.331,149.106
C08039=1147.083,42.853,-50.549,-179.851,6.332,149.105
C08040=1147.078,43.102,-50.565,-179.848,6.333,149.105
C08041=1147.073,43.352,-50.580,-179.846,6.334,149.104
C08042=1147.068,43.601,-50.595,-179.843,6.335,149.103
C08043=1147.063,43.851,-50.611,-179.841,6.336,149.103
C08044=1147.058,44.101,-50.626,-179.838,6.337,149.103
C08045=1147.053,44.350,-50.641,-179.835,6.338,149.102
C08046=1147.048,44.599,-50.656,-179.833,6.340,149.101
C08047=1147.042,44.849,-50.672,-179.830,6.340,149.101
C08048=1147.037,45.098,-50.687,-179.827,6.342,149.100
C08049=1147.033,45.348,-50.703,-179.825,6.343,149.100
C08050=1147.028,45.597,-50.718,-179.822,6.344,149.099
C08051=1147.023,45.846,-50.733,-179.820,6.345,149.099
C08052=1147.018,46.096,-50.749,-179.817,6.345,149.098
C08053=1147.012,46.345,-50.764,-179.814,6.347,149.098
C08054=1147.008,46.595,-50.780,-179.812,6.348,149.097
C08055=1147.003,46.844,-50.795,-179.809,6.349,149.097
C08056=1146.997,47.094,-50.811,-179.807,6.350,149.096
C08057=1146.992,47.343,-50.825,-179.804,6.351,149.096
C08058=1146.988,47.594,-50.841,-179.801,6.352,149.095
C08059=1146.982,47.843,-50.857,-179.799,6.353,149.095
C08060=1146.978,48.092,-50.872,-179.796,6.354,149.094
C08061=1146.973,48.341,-50.888,-179.793,6.356,149.093
C08062=1146.968,48.591,-50.904,-179.791,6.356,149.093
C08063=1146.962,48.840,-50.920,-179.788,6.358,149.092
C08064=1146.958,49.089,-50.935,-179.786,6.359,149.092
C08065=1146.952,49.339,-50.950,-179.782,6.360,149.091
C08066=1146.948,49.589,-50.966,-179.780,6.361,149.091
C08067=1146.943,49.838,-50.981,-179.778,6.362,149.090
C08068=1146.938,50.087,-50.997,-179.775,6.363,149.090
C08069=1146.932,50.337,-51.012,-179.772,6.364,149.089
C08070=1146.927,50.587,-51.028,-179.770,6.365,149.089
C08071=1146.923,50.836,-51.043,-179.767,6.367,149.088
C08072=1146.917,51.085,-51.059,-179.765,6.367,149.088
C08073=1146.913,51.335,-51.076,-179.761,6.369,149.087
C08074=1146.907,51.584,-51.091,-179.759,6.370,149.087
C08075=1146.902,51.834,-51.107,-179.756,6.371,149.086
C08076=1146.897,52.083,-51.122,-179.754,6.372,149.085
C08077=1146.893,52.333,-51.138,-179.751,6.373,149.085
C08078=1146.887,52.582,-51.153,-179.749,6.374,149.085
C08079=1146.882,52.831,-51.170,-179.746,6.375,149.084
C08080=1146.877,53.081,-51.186,-179.744,6.376,149.083
C08081=1146.872,53.350,-51.203,-179.740,6.378,149.083
C08082=1146.867,53.618,-51.219,-179.738,6.379,149.082
C08083=1146.861,53.886,-51.236,-179.735,6.380,149.082
C08084=1146.856,54.155,-51.253,-179.732,6.381,149.081
C08085=1146.851,54.405,-51.269,-179.730,6.382,149.081
C08086=1146.846,54.654,-51.285,-179.727,6.383,149.080
C08087=1146.841,54.904,-51.300,-179.724,6.385,149.080
C08088=1146.836,55.153,-51.317,-179.721,6.386,149.079
C08089=1146.830,55.403,-51.332,-179.719,6.387,149.079
C08090=1146.826,55.653,-51.348,-179.716,6.388,149.078
C08091=1146.820,55.902,-51.364,-179.713,6.389,149.077
C08092=1146.816,56.151,-51.380,-179.711,6.390,149.077
C08093=1146.811,56.401,-51.396,-179.708,6.391,149.076
C08094=1146.806,56.650,-51.411,-179.706,6.392,149.076
C08095=1146.801,56.900,-51.428,-179.703,6.394,149.075
C08096=1146.796,57.149,-51.443,-179.700,6.394,149.075
C08097=1146.791,57.398,-51.460,-179.698,6.396,149.074
C08098=1146.786,57.648,-51.476,-179.695,6.397,149.074
C08099=1146.781,57.897,-51.491,-179.692,6.398,149.073
C08100=1146.776,58.147,-51.508,-179.690,6.399,149.073
C08101=1146.771,58.396,-51.524,-179.687,6.401,149.072
C08102=1146.766,58.645,-51.540,-179.684,6.402,149.072
C08103=1146.761,58.895,-51.556,-179.682,6.403,149.071
C08104=1146.756,59.144,-51.571,-179.679,6.404,149.071
C08105=1146.751,59.394,-51.588,-179.676,6.405,149.070
C08106=1146.746,59.643,-51.604,-179.674,6.407,149.070
C08107=1146.741,59.893,-51.620,-179.671,6.407,149.069
C08108=1146.736,60.142,-51.636,-179.668,6.409,149.069
C08109=1146.731,60.392,-51.653,-179.666,6.410,149.068
C08110=1146.726,60.641,-51.668,-179.663,6.411,149.068
C08111=1146.721,60.890,-51.684,-179.660,6.413,149.067
C08112=1146.716,61.140,-51.700,-179.658,6.413,149.067
C08113=1146.711,61.389,-51.717,-179.655,6.415,149.066
C08114=1146.706,61.639,-51.733,-179.653,6.416,149.066
C08115=1146.701,61.888,-51.749,-179.650,6.417,149.065
C08116=1146.696,62.138,-51.765,-179.647,6.418,149.064
C08117=1146.691,62.387,-51.781,-179.645,6.419,149.064
C08118=1146.686,62.636,-51.798,-179.642,6.421,149.064
C08119=1146.681,62.886,-51.814,-179.639,6.422,149.063
C08120=1146.676,63.135,-51.831,-179.636,6.423,149.062
C08121=1146.671,63.385,-51.846,-179.634,6.424,149.062
C08122=1146.666,63.634,-51.863,-179.631,6.425,149.061
C08123=1146.661,63.883,-51.879,-179.628,6.427,149.061
C08124=1146.656,64.133,-51.895,-179.626,6.428,149.060
C08125=1146.651,64.382,-51.912,-179.623,6.429,149.060
C08126=1146.647,64.632,-51.928,-179.621,6.430,149.059
C08127=1146.641,64.882,-51.945,-179.618,6.432,149.059
C08128=1146.636,65.130,-51.961,-179.615,6.433,149.058
C08129=1146.632,65.380,-51.978,-179.613,6.434,149.058
C08130=1146.626,65.629,-51.993,-179.610,6.435,149.057
C08131=1146.622,65.879,-52.010,-179.607,6.436,149.057
C08132=1146.617,66.128,-52.026,-179.605,6.438,149.056
C08133=1146.611,66.378,-52.043,-179.602,6.439,149.056
C08134=1146.606,66.627,-52.059,-179.599,6.440,149.055
C08135=1146.602,66.876,-52.076,-179.596,6.441,149.055
C08136=1146.597,67.126,-52.093,-179.594,6.442,149.054
C08137=1146.592,67.375,-52.108,-179.591,6.444,149.054
C08138=1146.587,67.625,-52.125,-179.588,6.445,149.053
C08139=1146.582,67.874,-52.142,-179.586,6.446,149.053
C08140=1146.577,68.123,-52.158,-179.583,6.447,149.052
C08141=1146.573,68.373,-52.175,-179.581,6.448,149.052
C08142=1146.566,68.622,-52.191,-179.578,6.450,149.051
C08143=1146.562,68.872,-52.208,-179.575,6.451,149.051
C08144=1146.557,69.121,-52.224,-179.573,6.452,149.050
C08145=1146.552,69.370,-52.241,-179.570,6.454,149.050
C08146=1146.547,69.620,-52.258,-179.567,6.455,149.049
C08147=1146.542,69.869,-52.274,-179.564,6.456,149.049
C08148=1146.537,70.119,-52.290,-179.562,6.457,149.048
C08149=1146.533,70.368,-52.307,-179.560,6.458,149.048
C08150=1146.527,70.617,-52.324,-179.556,6.460,149.047
C08151=1146.523,70.867,-52.341,-179.554,6.461,149.047
C08152=1146.518,71.116,-52.357,-179.551,6.462,149.046
C08153=1146.512,71.366,-52.374,-179.548,6.463,149.046
C08154=1146.508,71.615,-52.391,-179.545,6.465,149.045
C08155=1146.503,71.865,-52.407,-179.543,6.466,149.045
C08156=1146.498,72.114,-52.424,-179.540,6.467,149.044
C08157=1146.493,72.363,-52.441,-179.537,6.469,149.044
C08158=1146.488,72.613,-52.458,-179.535,6.470,149.043
C08159=1146.483,72.862,-52.475,-179.532,6.471,149.043
C08160=1146.478,73.111,-52.491,-179.529,6.473,149.042
C08161=1146.473,73.361,-52.509,-179.527,6.474,149.042
C08162=1146.468,73.610,-52.525,-179.524,6.475,149.041
C08163=1146.463,73.859,-52.542,-179.521,6.477,149.041
C08164=1146.458,74.109,-52.559,-179.519,6.477,149.040
C08165=1146.453,74.358,-52.575,-179.516,6.479,149.040
C08166=1146.448,74.608,-52.592,-179.514,6.480,149.039
C08167=1146.443,74.857,-52.609,-179.511,6.481,149.039
C08168=1146.438,75.107,-52.626,-179.508,6.483,149.038
C08169=1146.433,75.356,-52.643,-179.505,6.483,149.038
C08170=1146.429,75.605,-52.659,-179.503,6.485,149.037
C08171=1146.423,75.855,-52.677,-179.500,6.487,149.037
C08172=1146.419,76.104,-52.693,-179.497,6.488,149.036
C08173=1146.413,76.354,-52.710,-179.495,6.489,149.036
C08174=1146.409,76.602,-52.727,-179.492,6.491,149.035
C08175=1146.404,76.852,-52.745,-179.489,6.492,149.035
C08176=1146.399,77.102,-52.761,-179.487,6.493,149.034
C08177=1146.393,77.351,-52.778,-179.484,6.494,149.034
C08178=1146.389,77.600,-52.795,-179.481,6.496,149.033
C08179=1146.384,77.850,-52.812,-179.479,6.497,149.033
C08180=1146.380,78.099,-52.830,-179.476,6.498,149.032
C08181=1146.374,78.348,-52.847,-179.473,6.500,149.032
C08182=1146.369,78.597,-52.863,-179.471,6.501,149.031
C08183=1146.364,78.847,-52.880,-179.468,6.502,149.031
C08184=1146.360,79.096,-52.898,-179.465,6.504,149.030
C08185=1146.354,79.364,-52.916,-179.462,6.505,149.030
C08186=1146.349,79.633,-52.935,-179.459,6.507,149.029
C08187=1146.344,79.902,-52.953,-179.457,6.508,149.029
C08188=1146.338,80.170,-52.971,-179.453,6.509,149.028
C08189=1146.333,80.420,-52.989,-179.451,6.510,149.028
C08190=1146.329,80.669,-53.006,-179.448,6.512,149.027
C08191=1146.323,80.918,-53.023,-179.445,6.514,149.027
C08192=1146.319,81.168,-53.040,-179.443,6.514,149.026
C08193=1146.313,81.416,-53.057,-179.440,6.516,149.026
C08194=1146.308,81.666,-53.075,-179.437,6.518,149.025
C08195=1146.304,81.916,-53.091,-179.435,6.518,149.025
C08196=1146.299,82.165,-53.109,-179.432,6.520,149.024
C08197=1146.294,82.414,-53.126,-179.429,6.521,149.024
C08198=1146.289,82.664,-53.143,-179.426,6.523,149.023
C08199=1146.284,82.913,-53.161,-179.424,6.524,149.023
C08200=1146.279,83.162,-53.178,-179.421,6.525,149.022
C08201=1146.274,83.411,-53.196,-179.418,6.527,149.022
C08202=1146.269,83.661,-53.213,-179.416,6.528,149.021
C08203=1146.264,83.910,-53.230,-179.413,6.529,149.021
C08204=1146.259,84.160,-53.248,-179.410,6.531,149.020
C08205=1146.254,84.409,-53.265,-179.407,6.533,149.020
C08206=1146.249,84.659,-53.283,-179.405,6.533,149.020
C08207=1146.245,84.908,-53.299,-179.402,6.535,149.019
C08208=1146.240,85.157,-53.317,-179.399,6.536,149.018
C08209=1146.235,85.407,-53.335,-179.397,6.538,149.018
C08210=1146.231,85.656,-53.352,-179.394,6.539,149.018
C08211=1146.225,85.905,-53.369,-179.391,6.540,149.017
C08212=1146.220,86.154,-53.387,-179.388,6.542,149.017
C08213=1146.215,86.404,-53.404,-179.386,6.544,149.016
C08214=1146.210,86.653,-53.422,-179.384,6.544,149.016
C08215=1146.205,86.903,-53.439,-179.380,6.546,149.015
C08216=1146.200,87.152,-53.457,-179.378,6.547,149.015
C08217=1146.195,87.401,-53.475,-179.375,6.549,149.014
C08218=1146.190,87.651,-53.492,-179.373,6.550,149.014
C08219=1146.186,87.900,-53.509,-179.369,6.551,149.013
C08220=1146.181,88.149,-53.527,-179.367,6.553,149.013
C08221=1146.176,88.399,-53.545,-179.364,6.555,149.012
C08222=1146.171,88.648,-53.563,-179.362,6.555,149.012
C08223=1146.166,88.898,-53.580,-179.359,6.557,149.011
C08224=1146.162,89.146,-53.597,-179.356,6.558,149.011
C08225=1146.157,89.396,-53.615,-179.353,6.560,149.010
C08226=1146.151,89.645,-53.633,-179.350,6.562,149.010
C08227=1146.147,89.895,-53.651,-179.348,6.562,149.009
C08228=1146.142,90.144,-53.669,-179.345,6.564,149.009
C08229=1146.136,90.394,-53.686,-179.342,6.566,149.008
C08230=1146.131,90.643,-53.704,-179.340,6.567,149.008
C08231=1146.127,90.892,-53.721,-179.337,6.568,149.008
C08232=1146.122,91.141,-53.739,-179.334,6.570,149.007
C08233=1146.117,91.391,-53.756,-179.332,6.571,149.007
C08234=1146.112,91.640,-53.774,-179.329,6.573,149.006
C08235=1146.107,91.889,-53.792,-179.326,6.575,149.006
C08236=1146.102,92.138,-53.810,-179.323,6.575,149.005
C08237=1146.097,92.388,-53.828,-179.321,6.577,149.005
C08238=1146.092,92.637,-53.846,-179.318,6.578,149.004
C08239=1146.087,92.886,-53.864,-179.315,6.580,149.004
C08240=1146.082,93.135,-53.882,-179.312,6.582,149.003
C08241=1146.078,93.385,-53.900,-179.310,6.582,149.003
C08242=1146.072,93.634,-53.917,-179.307,6.584,149.002
C08243=1146.068,93.884,-53.935,-179.304,6.586,149.002
C08244=1146.063,94.133,-53.953,-179.302,6.587,149.002
C08245=1146.059,94.382,-53.971,-179.298,6.589,149.001
C08246=1146.054,94.632,-53.988,-179.296,6.589,149.000
C08247=1146.049,94.881,-54.006,-179.294,6.591,149.000
C08248=1146.044,95.130,-54.024,-179.291,6.593,149.000
C08249=1146.039,95.379,-54.043,-179.288,6.595,148.999
C08250=1146.034,95.629,-54.061,-179.285,6.596,148.999
C08251=1146.029,95.878,-54.079,-179.283,6.597,148.998
C08252=1146.024,96.128,-54.096,-179.280,6.598,148.998
C08253=1146.019,96.377,-54.115,-179.277,6.600,148.997
C08254=1146.014,96.627,-54.133,-179.275,6.602,148.997
C08255=1146.009,96.876,-54.151,-179.271,6.603,148.996
C08256=1146.004,97.125,-54.169,-179.269,6.605,148.996
C08257=1146.000,97.374,-54.187,-179.266,6.606,148.995
C08258=1145.995,97.623,-54.204,-179.264,6.607,148.995
C08259=1145.990,97.872,-54.222,-179.261,6.609,148.995
C08260=1145.985,98.122,-54.241,-179.258,6.610,148.994
C08261=1145.981,98.371,-54.259,-179.255,6.612,148.994
C08262=1145.976,98.621,-54.277,-179.252,6.614,148.993
C08263=1145.971,98.869,-54.295,-179.250,6.615,148.993
C08264=1145.965,99.119,-54.314,-179.247,6.616,148.992
C08265=1145.960,99.368,-54.332,-179.244,6.618,148.992
C08266=1145.956,99.618,-54.350,-179.241,6.619,148.991
C08267=1145.951,99.867,-54.368,-179.239,6.621,148.991
C08268=1145.946,100.116,-54.386,-179.236,6.623,148.990
C08269=1145.941,100.365,-54.404,-179.233,6.624,148.990
C08270=1145.937,100.614,-54.422,-179.231,6.625,148.990
C08271=1145.931,100.865,-54.441,-179.228,6.626,148.989
C08272=1145.927,101.113,-54.460,-179.225,6.628,148.988
C08273=1145.922,101.362,-54.478,-179.222,6.630,148.988
C08274=1145.917,101.612,-54.496,-179.220,6.632,148.988
C08275=1145.912,101.861,-54.514,-179.217,6.633,148.987
C08276=1145.907,102.111,-54.533,-179.214,6.635,148.987
C08277=1145.902,102.359,-54.552,-179.212,6.635,148.986
C08278=1145.898,102.609,-54.569,-179.209,6.637,148.986
C08279=1145.893,102.858,-54.587,-179.206,6.639,148.985
C08280=1145.888,103.108,-54.606,-179.203,6.640,148.985
C08281=1145.883,103.357,-54.624,-179.201,6.642,148.985
C08282=1145.878,103.606,-54.643,-179.198,6.643,148.984
C08283=1145.873,103.855,-54.661,-179.195,6.645,148.983
C08284=1145.868,104.105,-54.680,-179.192,6.647,148.983
C08285=1145.863,104.354,-54.699,-179.190,6.648,148.983
C08286=1145.859,104.603,-54.717,-179.187,6.649,148.982
C08287=1145.854,104.853,-54.735,-179.184,6.651,148.982
C08288=1145.849,105.102,-54.754,-179.181,6.652,148.981
C08289=1145.844,105.370,-54.774,-179.179,6.654,148.981
C08290=1145.838,105.638,-54.794,-179.176,6.656,148.980
C08291=1145.833,105.907,-54.813,-179.173,6.657,148.980
C08292=1145.828,106.175,-54.834,-179.169,6.660,148.979
C08293=1145.823,106.424,-54.852,-179.167,6.660,148.979
C08294=1145.818,106.674,-54.870,-179.164,6.662,148.979
C08295=1145.813,106.923,-54.890,-179.162,6.664,148.978
C08296=1145.809,107.172,-54.908,-179.159,6.666,148.978
C08297=1145.804,107.421,-54.927,-179.156,6.667,148.977
C08298=1145.799,107.671,-54.945,-179.153,6.669,148.977
C08299=1145.794,107.920,-54.964,-179.150,6.670,148.976
C08300=1145.789,108.169,-54.982,-179.148,6.672,148.976
C08301=1145.784,108.419,-55.001,-179.145,6.674,148.975
C08302=1145.780,108.668,-55.020,-179.142,6.675,148.975
C08303=1145.774,108.917,-55.038,-179.139,6.677,148.975
C08304=1145.770,109.166,-55.057,-179.137,6.678,148.974
C08305=1145.765,109.416,-55.075,-179.134,6.679,148.974
C08306=1145.760,109.665,-55.095,-179.131,6.681,148.973
C08307=1145.756,109.914,-55.114,-179.129,6.683,148.973
C08308=1145.750,110.163,-55.132,-179.126,6.684,148.972
C08309=1145.746,110.412,-55.151,-179.123,6.686,148.972
C08310=1145.741,110.662,-55.170,-179.120,6.688,148.972
C08311=1145.736,110.911,-55.189,-179.118,6.689,148.971
C08312=1145.731,111.161,-55.208,-179.114,6.691,148.970
C08313=1145.726,111.409,-55.226,-179.112,6.692,148.970
C08314=1145.721,111.659,-55.246,-179.109,6.694,148.970
C08315=1145.717,111.908,-55.264,-179.106,6.696,148.969
C08316=1145.712,112.158,-55.284,-179.104,6.697,148.969
C08317=1145.707,112.407,-55.302,-179.101,6.699,148.968
C08318=1145.702,112.656,-55.321,-179.098,6.701,148.968
C08319=1145.698,112.905,-55.340,-179.096,6.702,148.968
C08320=1145.692,113.154,-55.358,-179.093,6.703,148.967
C08321=1145.688,113.404,-55.378,-179.090,6.705,148.967
C08322=1145.683,113.652,-55.397,-179.087,6.706,148.966
C08323=1145.679,113.902,-55.416,-179.085,6.708,148.966
C08324=1145.673,114.151,-55.434,-179.082,6.710,148.965
C08325=1145.668,114.401,-55.454,-179.079,6.711,148.965
C08326=1145.664,114.649,-55.473,-179.076,6.713,148.965
C08327=1145.659,114.899,-55.492,-179.074,6.715,148.964
C08328=1145.654,115.148,-55.510,-179.071,6.717,148.964
C08329=1145.649,115.398,-55.530,-179.068,6.718,148.963
C08330=1145.644,115.646,-55.549,-179.065,6.720,148.963
C08331=1145.640,115.896,-55.568,-179.062,6.721,148.962
C08332=1145.634,116.145,-55.587,-179.060,6.723,148.962
C08333=1145.630,116.394,-55.606,-179.057,6.725,148.961
C08334=1145.625,116.643,-55.625,-179.054,6.726,148.961
C08335=1145.620,116.893,-55.645,-179.051,6.728,148.961
C08336=1145.615,117.141,-55.664,-179.049,6.730,148.960
C08337=1145.611,117.391,-55.683,-179.046,6.731,148.960
C08338=1145.605,117.640,-55.703,-179.043,6.733,148.959
C08339=1145.601,117.890,-55.721,-179.040,6.735,148.959
C08340=1145.596,118.139,-55.740,-179.038,6.737,148.959
C08341=1145.591,118.388,-55.760,-179.035,6.738,148.958
C08342=1145.586,118.637,-55.779,-179.032,6.740,148.958
C08343=1145.582,118.886,-55.798,-179.029,6.741,148.957
C08344=1145.576,119.135,-55.818,-179.026,6.743,148.957
C08345=1145.572,119.385,-55.837,-179.024,6.745,148.956
C08346=1145.568,119.634,-55.856,-179.021,6.746,148.956
C08347=1145.562,119.883,-55.876,-179.018,6.748,148.956
C08348=1145.557,120.132,-55.895,-179.016,6.750,148.955
C08349=1145.552,120.381,-55.915,-179.013,6.751,148.955
C08350=1145.548,120.631,-55.934,-179.010,6.753,148.954
C08351=1145.543,120.879,-55.953,-179.007,6.755,148.954
C08352=1145.538,121.129,-55.973,-179.005,6.757,148.954
C08353=1145.533,121.379,-55.992,-179.002,6.758,148.953
C08354=1145.528,121.627,-56.012,-178.999,6.760,148.953
C08355=1145.524,121.877,-56.031,-178.996,6.761,148.952
C08356=1145.519,122.126,-56.050,-178.993,6.763,148.952
C08357=1145.514,122.375,-56.070,-178.991,6.765,148.951
C08358=1145.509,122.625,-56.089,-178.988,6.766,148.951
C08359=1145.504,122.874,-56.108,-178.985,6.768,148.951
C08360=1145.500,123.122,-56.128,-178.982,6.770,148.950
C08361=1145.495,123.372,-56.148,-178.980,6.771,148.950
C08362=1145.490,123.621,-56.167,-178.977,6.773,148.949
C08363=1145.485,123.870,-56.187,-178.974,6.775,148.949
C08364=1145.480,124.120,-56.207,-178.971,6.777,148.949
C08365=1145.475,124.369,-56.226,-178.969,6.778,148.948
C08366=1145.471,124.618,-56.246,-178.966,6.780,148.948
C08367=1145.467,124.867,-56.265,-178.963,6.782,148.947
C08368=1145.461,125.116,-56.285,-178.961,6.783,148.947
C08369=1145.457,125.365,-56.304,-178.958,6.785,148.947
C08370=1145.452,125.615,-56.324,-178.955,6.787,148.946
C08371=1145.447,125.864,-56.344,-178.952,6.788,148.946
C08372=1145.442,126.113,-56.364,-178.950,6.790,148.945
C08373=1145.437,126.362,-56.383,-178.947,6.792,148.945
C08374=1145.433,126.612,-56.403,-178.944,6.794,148.945
C08375=1145.428,126.860,-56.423,-178.940,6.796,148.944
C08376=1145.423,127.110,-56.442,-178.938,6.797,148.944
C08377=1145.418,127.359,-56.462,-178.935,6.799,148.943
C08378=1145.414,127.608,-56.483,-178.932,6.801,148.943
C08379=1145.408,127.857,-56.502,-178.930,6.802,148.942
C08380=1145.404,128.107,-56.521,-178.927,6.804,148.942
C08381=1145.399,128.356,-56.542,-178.924,6.806,148.942
C08382=1145.394,128.605,-56.561,-178.921,6.808,148.941
C08383=1145.389,128.854,-56.581,-178.919,6.809,148.941
C08384=1145.385,129.103,-56.601,-178.916,6.811,148.940
C08385=1145.380,129.353,-56.621,-178.913,6.813,148.940
C08386=1145.375,129.601,-56.641,-178.911,6.814,148.940
C08387=1145.370,129.850,-56.660,-178.908,6.816,148.939
C08388=1145.366,130.099,-56.681,-178.905,6.818,148.939
C08389=1145.361,130.349,-56.700,-178.902,6.820,148.938
C08390=1145.356,130.598,-56.720,-178.899,6.822,148.938
C08391=1145.351,130.847,-56.740,-178.896,6.824,148.938
C08392=1145.346,131.096,-56.760,-178.894,6.825,148.937
C08393=1145.341,131.365,-56.782,-178.891,6.827,148.937
C08394=1145.336,131.633,-56.803,-178.888,6.829,148.936
C08395=1145.331,131.902,-56.824,-178.885,6.831,148.936
C08396=1145.326,132.170,-56.847,-178.882,6.833,148.936
C08397=1145.321,132.420,-56.866,-178.879,6.835,148.935
C08398=1145.317,132.669,-56.887,-178.877,6.836,148.935
C08399=1145.312,132.918,-56.906,-178.874,6.838,148.935
C08400=1145.307,133.167,-56.926,-178.871,6.841,148.934
C08401=1145.301,133.416,-56.947,-178.868,6.842,148.934
C08402=1145.297,133.665,-56.967,-178.865,6.844,148.933
C08403=1145.293,133.914,-56.987,-178.863,6.846,148.933
C08404=1145.288,134.164,-57.007,-178.860,6.847,148.933
C08405=1145.283,134.413,-57.027,-178.857,6.849,148.932
C08406=1145.278,134.662,-57.048,-178.854,6.851,148.932
C08407=1145.273,134.911,-57.068,-178.852,6.853,148.931
C08408=1145.268,135.160,-57.088,-178.849,6.854,148.931
C08409=1145.264,135.409,-57.108,-178.846,6.857,148.931
C08410=1145.259,135.658,-57.128,-178.843,6.859,148.930
C08411=1145.254,135.908,-57.149,-178.840,6.860,148.930
C08412=1145.250,136.157,-57.169,-178.838,6.862,148.929
C08413=1145.245,136.406,-57.189,-178.835,6.864,148.929
C08414=1145.240,136.655,-57.210,-178.832,6.865,148.929
C08415=1145.235,136.904,-57.230,-178.829,6.867,148.928
C08416=1145.230,137.153,-57.250,-178.827,6.869,148.928
C08417=1145.225,137.402,-57.270,-178.823,6.871,148.927
C08418=1145.221,137.651,-57.291,-178.821,6.873,148.927
C08419=1145.216,137.900,-57.311,-178.818,6.875,148.927
C08420=1145.211,138.149,-57.332,-178.815,6.876,148.926
C08421=1145.207,138.399,-57.352,-178.813,6.878,148.926
C08422=1145.202,138.648,-57.372,-178.810,6.880,148.926
C08423=1145.197,138.897,-57.393,-178.807,6.882,148.925
C08424=1145.193,139.146,-57.413,-178.804,6.884,148.925
C08425=1145.187,139.395,-57.434,-178.801,6.886,148.924
C08426=1145.183,139.644,-57.455,-178.798,6.887,148.924
C08427=1145.179,139.893,-57.475,-178.796,6.890,148.924
C08428=1145.173,140.143,-57.496,-178.793,6.891,148.923
C08429=1145.169,140.392,-57.516,-178.791,6.893,148.923
C08430=1145.164,140.641,-57.536,-178.788,6.895,148.923
C08431=1145.159,140.890,-57.557,-178.785,6.897,148.922
C08432=1145.155,141.139,-57.577,-178.782,6.899,148.922
C08433=1145.149,141.389,-57.598,-178.779,6.901,148.921
C08434=1145.145,141.637,-57.619,-178.777,6.902,148.921
C08435=1145.141,141.886,-57.639,-178.774,6.904,148.921
C08436=1145.135,142.136,-57.660,-178.771,6.906,148.920
C08437=1145.131,142.385,-57.680,-178.768,6.908,148.920
C08438=1145.126,142.634,-57.701,-178.765,6.910,148.920
C08439=1145.121,142.883,-57.722,-178.762,6.912,148.919
C08440=1145.117,143.132,-57.742,-178.760,6.913,148.919
C08441=1145.112,143.381,-57.763,-178.757,6.915,148.918
C08442=1145.107,143.630,-57.783,-178.754,6.918,148.918
C08443=1145.102,143.879,-57.804,-178.751,6.920,148.918
C08444=1145.098,144.128,-57.825,-178.749,6.921,148.917
C08445=1145.093,144.377,-57.846,-178.746,6.923,148.917
C08446=1145.088,144.626,-57.867,-178.743,6.925,148.917
C08447=1145.084,144.876,-57.888,-178.740,6.927,148.916
C08448=1145.079,145.125,-57.908,-178.737,6.929,148.916
C08449=1145.074,145.374,-57.929,-178.735,6.931,148.916
C08450=1145.070,145.623,-57.950,-178.732,6.932,148.915
C08451=1145.065,145.872,-57.971,-178.729,6.934,148.915
C08452=1145.059,146.121,-57.992,-178.726,6.936,148.914
C08453=1145.055,146.370,-58.013,-178.724,6.939,148.914
C08454=1145.050,146.619,-58.034,-178.721,6.941,148.914
C08455=1145.046,146.868,-58.054,-178.718,6.942,148.913
C08456=1145.040,147.117,-58.075,-178.715,6.944,148.913
C08457=1145.037,147.367,-58.096,-178.712,6.946,148.913
C08458=1145.032,147.615,-58.118,-178.709,6.948,148.912
C08459=1145.027,147.865,-58.139,-178.707,6.950,148.912
C08460=1145.022,148.114,-58.159,-178.704,6.952,148.912
C08461=1145.017,148.363,-58.180,-178.701,6.953,148.911
C08462=1145.013,148.611,-58.201,-178.698,6.956,148.911
C08463=1145.008,148.861,-58.222,-178.696,6.958,148.911
C08464=1145.003,149.111,-58.243,-178.693,6.960,148.910
C08465=1144.999,149.359,-58.264,-178.690,6.961,148.910
C08466=1144.994,149.608,-58.285,-178.687,6.964,148.910
C08467=1144.989,149.857,-58.306,-178.684,6.966,148.909
C08468=1144.985,150.106,-58.327,-178.682,6.967,148.909
C08469=1144.979,150.355,-58.348,-178.679,6.969,148.908
C08470=1144.975,150.605,-58.370,-178.677,6.971,148.908
C08471=1144.971,150.853,-58.391,-178.673,6.974,148.908
C08472=1144.965,151.103,-58.412,-178.671,6.975,148.907
C08473=1144.961,151.351,-58.433,-178.668,6.977,148.907
C08474=1144.955,151.600,-58.454,-178.665,6.979,148.907
C08475=1144.952,151.850,-58.475,-178.662,6.981,148.906
C08476=1144.947,152.099,-58.497,-178.659,6.983,148.906
C08477=1144.942,152.348,-58.518,-178.657,6.985,148.906
C08478=1144.937,152.597,-58.539,-178.654,6.987,148.905
C08479=1144.932,152.846,-58.560,-178.651,6.989,148.905
C08480=1144.928,153.095,-58.582,-178.648,6.991,148.905
C08481=1144.923,153.344,-58.603,-178.646,6.993,148.904
C08482=1144.918,153.593,-58.624,-178.643,6.994,148.904
C08483=1144.913,153.842,-58.645,-178.640,6.997,148.904
C08484=1144.909,154.091,-58.667,-178.637,6.999,148.903
C08485=1144.904,154.340,-58.688,-178.635,7.001,148.903
C08486=1144.899,154.589,-58.710,-178.631,7.003,148.903
C08487=1144.895,154.838,-58.732,-178.629,7.005,148.902
C08488=1144.890,155.088,-58.753,-178.626,7.007,148.902
C08489=1144.886,155.336,-58.774,-178.623,7.008,148.901
C08490=1144.880,155.585,-58.795,-178.620,7.011,148.901
C08491=1144.876,155.835,-58.817,-178.618,7.013,148.901
C08492=1144.871,156.083,-58.838,-178.615,7.015,148.901
C08493=1144.866,156.332,-58.859,-178.612,7.017,148.900
C08494=1144.862,156.582,-58.881,-178.609,7.019,148.900
C08495=1144.857,156.830,-58.903,-178.607,7.021,148.900
C08496=1144.852,157.080,-58.924,-178.604,7.023,148.899
C08497=1144.847,157.348,-58.947,-178.601,7.025,148.899
C08498=1144.842,157.617,-58.971,-178.598,7.027,148.899
C08499=1144.837,157.886,-58.994,-178.595,7.030,148.898
C08500=1144.832,158.155,-59.018,-178.591,7.032,148.898
C08501=1144.827,158.404,-59.039,-178.589,7.034,148.897
C08502=1144.822,158.654,-59.061,-178.586,7.036,148.897
C08503=1144.818,158.902,-59.082,-178.583,7.037,148.897
C08504=1144.813,159.151,-59.103,-178.581,7.040,148.897
C08505=1144.809,159.401,-59.125,-178.578,7.042,148.896
C08506=1144.804,159.649,-59.146,-178.575,7.044,148.896
C08507=1144.800,159.899,-59.169,-178.572,7.046,148.895
C08508=1144.795,160.147,-59.190,-178.569,7.048,148.895
C08509=1144.790,160.396,-59.212,-178.567,7.050,148.895
C08510=1144.786,160.645,-59.234,-178.564,7.053,148.895
C08511=1144.781,160.895,-59.255,-178.561,7.054,148.894
C08512=1144.776,161.144,-59.277,-178.558,7.056,148.894
C08513=1144.771,161.393,-59.299,-178.555,7.059,148.894
C08514=1144.767,161.641,-59.320,-178.553,7.061,148.893
C08515=1144.762,161.891,-59.343,-178.550,7.062,148.893
C08516=1144.757,162.140,-59.365,-178.547,7.065,148.893
C08517=1144.752,162.389,-59.387,-178.544,7.067,148.892
C08518=1144.748,162.638,-59.408,-178.542,7.069,148.892
C08519=1144.743,162.887,-59.430,-178.538,7.071,148.892
C08520=1144.738,163.135,-59.452,-178.536,7.073,148.891
C08521=1144.734,163.384,-59.474,-178.533,7.075,148.891
C08522=1144.729,163.633,-59.496,-178.530,7.078,148.891
C08523=1144.724,163.882,-59.518,-178.528,7.079,148.890
C08524=1144.720,164.131,-59.540,-178.525,7.081,148.890
C08525=1144.715,164.380,-59.561,-178.522,7.083,148.890
C08526=1144.710,164.630,-59.584,-178.519,7.086,148.890
C08527=1144.705,164.878,-59.606,-178.517,7.087,148.889
C08528=1144.701,165.128,-59.628,-178.513,7.090,148.889
C08529=1144.696,165.376,-59.649,-178.511,7.092,148.888
C08530=1144.692,165.626,-59.671,-178.508,7.094,148.888
C08531=1144.687,165.874,-59.693,-178.505,7.096,148.888
C08532=1144.683,166.124,-59.715,-178.502,7.098,148.888
C08533=1144.678,166.372,-59.738,-178.500,7.100,148.887
C08534=1144.673,166.621,-59.760,-178.497,7.103,148.887
C08535=1144.668,166.870,-59.782,-178.494,7.104,148.887
C08536=1144.664,167.119,-59.804,-178.491,7.107,148.886
C08537=1144.659,167.368,-59.826,-178.488,7.108,148.886
C08538=1144.654,167.618,-59.848,-178.486,7.111,148.886
C08539=1144.650,167.866,-59.871,-178.483,7.113,148.885
C08540=1144.645,168.115,-59.893,-178.480,7.115,148.885
C08541=1144.640,168.365,-59.915,-178.477,7.117,148.885
C08542=1144.636,168.613,-59.937,-178.474,7.119,148.885
C08543=1144.631,168.863,-59.959,-178.472,7.121,148.884
C08544=1144.627,169.111,-59.981,-178.468,7.124,148.884
C08545=1144.622,169.360,-60.004,-178.466,7.126,148.884
C08546=1144.617,169.609,-60.026,-178.464,7.128,148.883
C08547=1144.613,169.858,-60.049,-178.460,7.130,148.883
C08548=1144.608,170.107,-60.071,-178.458,7.132,148.883
C08549=1144.603,170.356,-60.093,-178.455,7.134,148.882
C08550=1144.599,170.605,-60.116,-178.452,7.136,148.882
C08551=1144.593,170.854,-60.138,-178.449,7.138,148.882
C08552=1144.589,171.103,-60.160,-178.446,7.141,148.882
C08553=1144.585,171.352,-60.183,-178.444,7.143,148.881
C08554=1144.580,171.601,-60.205,-178.441,7.144,148.881
C08555=1144.575,171.850,-60.227,-178.438,7.147,148.880
C08556=1144.570,172.098,-60.250,-178.436,7.149,148.880
C08557=1144.566,172.348,-60.272,-178.432,7.152,148.880
C08558=1144.562,172.596,-60.295,-178.430,7.153,148.880
C08559=1144.556,172.845,-60.317,-178.427,7.156,148.879
C08560=1144.552,173.094,-60.340,-178.424,7.158,148.879
C08561=1144.547,173.344,-60.363,-178.421,7.160,148.879
C08562=1144.542,173.592,-60.384,-178.419,7.163,148.879
C08563=1144.538,173.841,-60.407,-178.416,7.164,148.878
C08564=1144.533,174.091,-60.430,-178.413,7.167,148.878
C08565=1144.529,174.339,-60.452,-178.410,7.169,148.878
C08566=1144.524,174.588,-60.475,-178.408,7.171,148.877
C08567=1144.520,174.837,-60.497,-178.404,7.173,148.877
C08568=1144.515,175.085,-60.520,-178.402,7.175,148.877
C08569=1144.510,175.335,-60.542,-178.399,7.178,148.877
C08570=1144.506,175.584,-60.566,-178.396,7.180,148.876
C08571=1144.501,175.832,-60.587,-178.393,7.183,148.876
C08572=1144.496,176.081,-60.611,-178.391,7.184,148.876
C08573=1144.492,176.330,-60.634,-178.387,7.187,148.875
C08574=1144.487,176.580,-60.656,-178.385,7.189,148.875
C08575=1144.483,176.828,-60.679,-178.382,7.191,148.875
C08576=1144.478,177.078,-60.701,-178.379,7.193,148.874
C08577=1144.474,177.326,-60.724,-178.377,7.195,148.874
C08578=1144.469,177.575,-60.747,-178.374,7.198,148.874
C08579=1144.463,177.824,-60.770,-178.371,7.199,148.874
C08580=1144.459,178.073,-60.792,-178.368,7.202,148.873
C08581=1144.455,178.322,-60.816,-178.365,7.204,148.873
C08582=1144.451,178.571,-60.839,-178.362,7.207,148.873
C08583=1144.445,178.820,-60.861,-178.360,7.209,148.873
C08584=1144.441,179.068,-60.884,-178.357,7.210,148.872
C08585=1144.436,179.317,-60.907,-178.354,7.213,148.872
C08586=1144.432,179.566,-60.930,-178.352,7.215,148.872
C08587=1144.427,179.816,-60.952,-178.348,7.218,148.871
C08588=1144.422,180.064,-60.975,-178.346,7.220,148.871
C08589=1144.417,180.313,-60.999,-178.343,7.222,148.871
C08590=1144.413,180.562,-61.021,-178.340,7.224,148.871
C08591=1144.409,180.811,-61.045,-178.337,7.227,148.870
C08592=1144.404,181.060,-61.068,-178.335,7.229,148.870
C08593=1144.399,181.309,-61.090,-178.332,7.232,148.870
C08594=1144.394,181.558,-61.113,-178.329,7.233,148.870
C08595=1144.390,181.807,-61.137,-178.326,7.236,148.869
C08596=1144.386,182.055,-61.159,-178.324,7.238,148.869
C08597=1144.381,182.304,-61.183,-178.320,7.240,148.869
C08598=1144.376,182.553,-61.206,-178.318,7.243,148.869
C08599=1144.372,182.802,-61.229,-178.315,7.245,148.868
C08600=1144.367,183.050,-61.252,-178.312,7.247,148.868
C08601=1144.362,183.321,-61.277,-178.309,7.250,148.868
C08602=1144.357,183.591,-61.302,-178.306,7.252,148.867
C08603=1144.353,183.860,-61.327,-178.303,7.254,148.867
C08604=1144.348,184.129,-61.352,-178.300,7.257,148.867
C08605=1144.343,184.378,-61.376,-178.297,7.259,148.867
C08606=1144.338,184.627,-61.399,-178.295,7.261,148.866
C08607=1144.333,184.876,-61.423,-178.292,7.264,148.866
C08608=1144.329,185.124,-61.445,-178.289,7.266,148.866
C08609=1144.324,185.373,-61.468,-178.286,7.268,148.865
C08610=1144.319,185.622,-61.492,-178.284,7.270,148.865
C08611=1144.315,185.872,-61.515,-178.280,7.273,148.865
C08612=1144.310,186.121,-61.538,-178.278,7.275,148.865
C08613=1144.305,186.370,-61.562,-178.275,7.278,148.865
C08614=1144.301,186.618,-61.585,-178.273,7.280,148.864
C08615=1144.297,186.867,-61.608,-178.269,7.282,148.864
C08616=1144.292,187.116,-61.632,-178.267,7.284,148.864
C08617=1144.288,187.365,-61.655,-178.264,7.287,148.864
C08618=1144.283,187.614,-61.679,-178.261,7.289,148.863
C08619=1144.278,187.863,-61.702,-178.258,7.292,148.863
C08620=1144.273,188.112,-61.725,-178.255,7.294,148.863
C08621=1144.269,188.360,-61.749,-178.253,7.296,148.863
C08622=1144.264,188.609,-61.773,-178.250,7.299,148.862
C08623=1144.260,188.858,-61.796,-178.247,7.301,148.862
C08624=1144.255,189.107,-61.820,-178.244,7.303,148.862
C08625=1144.250,189.356,-61.843,-178.242,7.305,148.862
C08626=1144.247,189.605,-61.866,-178.239,7.308,148.861
C08627=1144.242,189.854,-61.890,-178.236,7.310,148.861
C08628=1144.237,190.103,-61.913,-178.233,7.313,148.861
C08629=1144.233,190.351,-61.937,-178.230,7.314,148.860
C08630=1144.228,190.600,-61.961,-178.228,7.317,148.860
C08631=1144.223,190.849,-61.984,-178.224,7.320,148.860
C08632=1144.219,191.097,-62.008,-178.222,7.322,148.860
C08633=1144.214,191.347,-62.031,-178.219,7.325,148.860
C08634=1144.210,191.596,-62.055,-178.217,7.327,148.859
C08635=1144.205,191.844,-62.079,-178.213,7.329,148.859
C08636=1144.200,192.093,-62.103,-178.211,7.331,148.859
C08637=1144.195,192.342,-62.127,-178.208,7.334,148.859
C08638=1144.191,192.591,-62.150,-178.206,7.336,148.858
C08639=1144.186,192.840,-62.173,-178.202,7.338,148.858
C08640=1144.182,193.088,-62.198,-178.199,7.341,148.858
C08641=1144.177,193.337,-62.221,-178.197,7.343,148.858
C08642=1144.173,193.586,-62.245,-178.194,7.346,148.858
C08643=1144.168,193.835,-62.268,-178.191,7.348,148.857
C08644=1144.163,194.083,-62.292,-178.188,7.351,148.857
C08645=1144.159,194.332,-62.316,-178.185,7.353,148.857
C08646=1144.155,194.581,-62.340,-178.183,7.355,148.857
C08647=1144.150,194.831,-62.364,-178.180,7.358,148.856
C08648=1144.145,195.079,-62.388,-178.177,7.360,148.856
C08649=1144.140,195.328,-62.412,-178.174,7.362,148.856
C08650=1144.136,195.576,-62.436,-178.172,7.365,148.856
C08651=1144.132,195.825,-62.460,-178.169,7.367,148.855
C08652=1144.127,196.074,-62.483,-178.166,7.370,148.855
C08653=1144.122,196.323,-62.508,-178.163,7.372,148.855
C08654=1144.118,196.572,-62.532,-178.160,7.375,148.855
C08655=1144.113,196.821,-62.556,-178.158,7.376,148.854
C08656=1144.109,197.069,-62.580,-178.155,7.379,148.854
C08657=1144.104,197.318,-62.603,-178.152,7.382,148.854
C08658=1144.099,197.567,-62.628,-178.149,7.384,148.854
C08659=1144.095,197.815,-62.652,-178.147,7.387,148.854
C08660=1144.091,198.065,-62.675,-178.144,7.389,148.853
C08661=1144.086,198.313,-62.700,-178.141,7.391,148.853
C08662=1144.081,198.562,-62.724,-178.138,7.394,148.853
C08663=1144.077,198.811,-62.748,-178.136,7.396,148.853
C08664=1144.072,199.060,-62.772,-178.132,7.399,148.852
C08665=1144.068,199.309,-62.796,-178.130,7.402,148.852
C08666=1144.063,199.557,-62.821,-178.127,7.403,148.852
C08667=1144.059,199.806,-62.845,-178.124,7.406,148.852
C08668=1144.054,200.055,-62.868,-178.122,7.408,148.852
C08669=1144.049,200.304,-62.893,-178.119,7.411,148.851
C08670=1144.045,200.553,-62.917,-178.116,7.414,148.851
C08671=1144.041,200.801,-62.941,-178.113,7.416,148.851
C08672=1144.036,201.050,-62.966,-178.110,7.418,148.851
C08673=1144.031,201.298,-62.990,-178.107,7.421,148.851
C08674=1144.027,201.547,-63.015,-178.105,7.423,148.850
C08675=1144.022,201.797,-63.039,-178.102,7.426,148.850
C08676=1144.017,202.045,-63.063,-178.099,7.429,148.850
C08677=1144.013,202.294,-63.087,-178.096,7.431,148.850
C08678=1144.009,202.543,-63.112,-178.093,7.433,148.850
C08679=1144.004,202.791,-63.136,-178.091,7.435,148.849
C08680=1143.999,203.040,-63.160,-178.088,7.438,148.849
C08681=1143.995,203.289,-63.185,-178.085,7.441,148.849
C08682=1143.991,203.538,-63.209,-178.083,7.443,148.849
C08683=1143.986,203.786,-63.234,-178.079,7.445,148.849
C08684=1143.982,204.036,-63.258,-178.077,7.448,148.848
C08685=1143.977,204.284,-63.283,-178.074,7.450,148.848
C08686=1143.972,204.533,-63.307,-178.071,7.453,148.848
C08687=1143.967,204.781,-63.332,-178.068,7.456,148.848
C08688=1143.963,205.030,-63.356,-178.066,7.458,148.848
C08689=1143.958,205.279,-63.381,-178.063,7.461,148.847
C08690=1143.954,205.528,-63.405,-178.060,7.463,148.847
C08691=1143.949,205.777,-63.430,-178.057,7.465,148.847
C08692=1143.945,206.025,-63.455,-178.055,7.468,148.847
C08693=1143.940,206.274,-63.479,-178.051,7.471,148.847
C08694=1143.936,206.523,-63.504,-178.049,7.473,148.846
C08695=1143.931,206.771,-63.528,-178.046,7.476,148.846
C08696=1143.927,207.021,-63.553,-178.043,7.478,148.846
C08697=1143.922,207.269,-63.577,-178.041,7.480,148.846
C08698=1143.917,207.518,-63.602,-178.038,7.483,148.846
C08699=1143.914,207.766,-63.627,-178.035,7.486,148.845
C08700=1143.909,208.015,-63.652,-178.032,7.489,148.845
C08701=1143.904,208.264,-63.676,-178.029,7.490,148.845
C08702=1143.900,208.513,-63.701,-178.026,7.493,148.845
C08703=1143.896,208.761,-63.726,-178.024,7.496,148.845
C08704=1143.891,209.010,-63.751,-178.021,7.498,148.844
C08705=1143.886,209.280,-63.778,-178.018,7.501,148.844
C08706=1143.881,209.551,-63.805,-178.015,7.504,148.844
C08707=1143.875,209.822,-63.832,-178.012,7.506,148.844
C08708=1143.871,210.093,-63.859,-178.009,7.509,148.844
C08709=1143.867,210.341,-63.883,-178.006,7.512,148.843
C08710=1143.862,210.590,-63.908,-178.003,7.515,148.843
C08711=1143.857,210.839,-63.934,-178.000,7.518,148.843
C08712=1143.853,211.088,-63.958,-177.998,7.519,148.843
C08713=1143.849,211.336,-63.983,-177.995,7.522,148.843
C08714=1143.844,211.585,-64.008,-177.992,7.525,148.843
C08715=1143.840,211.834,-64.032,-177.989,7.527,148.842
C08716=1143.835,212.082,-64.058,-177.987,7.530,148.842
C08717=1143.830,212.331,-64.083,-177.984,7.533,148.842
C08718=1143.825,212.579,-64.108,-177.980,7.535,148.842
C08719=1143.822,212.828,-64.133,-177.978,7.537,148.842
C08720=1143.817,213.076,-64.158,-177.975,7.540,148.842
C08721=1143.812,213.326,-64.183,-177.972,7.543,148.841
C08722=1143.807,213.574,-64.208,-177.969,7.546,148.841
C08723=1143.804,213.823,-64.233,-177.967,7.548,148.841
C08724=1143.799,214.071,-64.258,-177.964,7.551,148.841
C08725=1143.794,214.321,-64.283,-177.961,7.553,148.841
C08726=1143.790,214.569,-64.309,-177.959,7.556,148.841
C08727=1143.785,214.818,-64.334,-177.956,7.558,148.840
C08728=1143.781,215.067,-64.359,-177.953,7.561,148.840
C08729=1143.776,215.315,-64.384,-177.950,7.564,148.840
C08730=1143.772,215.564,-64.409,-177.948,7.566,148.840
C08731=1143.767,215.812,-64.435,-177.945,7.569,148.840
C08732=1143.763,216.062,-64.460,-177.942,7.572,148.840
C08733=1143.758,216.310,-64.485,-177.939,7.574,148.839
C08734=1143.754,216.559,-64.511,-177.937,7.577,148.839
C08735=1143.750,216.808,-64.535,-177.933,7.579,148.839
C08736=1143.745,217.056,-64.561,-177.931,7.582,148.839
C08737=1143.741,217.305,-64.586,-177.928,7.585,148.839
C08738=1143.736,217.553,-64.611,-177.925,7.588,148.839
C08739=1143.731,217.802,-64.637,-177.922,7.590,148.838
C08740=1143.727,218.051,-64.663,-177.920,7.592,148.838
C08741=1143.722,218.299,-64.688,-177.917,7.595,148.838
C08742=1143.718,218.549,-64.713,-177.914,7.598,148.838
C08743=1143.713,218.797,-64.738,-177.911,7.600,148.838
C08744=1143.709,219.045,-64.764,-177.909,7.603,148.838
C08745=1143.705,219.294,-64.790,-177.906,7.606,148.838
C08746=1143.700,219.543,-64.815,-177.903,7.609,148.837
C08747=1143.695,219.792,-64.840,-177.900,7.611,148.837
C08748=1143.691,220.041,-64.866,-177.897,7.613,148.837
C08749=1143.686,220.289,-64.892,-177.895,7.616,148.837
C08750=1143.682,220.537,-64.917,-177.892,7.619,148.837
C08751=1143.678,220.786,-64.943,-177.889,7.622,148.837
C08752=1143.673,221.034,-64.968,-177.886,7.624,148.836
C08753=1143.669,221.283,-64.994,-177.884,7.627,148.836
C08754=1143.664,221.533,-65.019,-177.881,7.630,148.836
C08755=1143.659,221.781,-65.045,-177.878,7.633,148.836
C08756=1143.655,222.030,-65.070,-177.875,7.635,148.836
C08757=1143.651,222.278,-65.096,-177.872,7.637,148.836
C08758=1143.646,222.526,-65.121,-177.870,7.640,148.836
C08759=1143.642,222.775,-65.147,-177.867,7.643,148.836
C08760=1143.638,223.024,-65.173,-177.864,7.646,148.835
C08761=1143.633,223.273,-65.199,-177.861,7.649,148.835
C08762=1143.629,223.521,-65.224,-177.859,7.651,148.835
C08763=1143.624,223.770,-65.250,-177.856,7.654,148.835
C08764=1143.619,224.019,-65.276,-177.853,7.657,148.835
C08765=1143.615,224.267,-65.302,-177.850,7.660,148.835
C08766=1143.610,224.516,-65.327,-177.847,7.662,148.834
C08767=1143.606,224.764,-65.354,-177.844,7.665,148.834
C08768=1143.602,225.013,-65.380,-177.842,7.667,148.834
C08769=1143.597,225.261,-65.405,-177.839,7.670,148.834
C08770=1143.592,225.510,-65.431,-177.836,7.673,148.834
C08771=1143.588,225.759,-65.457,-177.833,7.676,148.834
C08772=1143.584,226.008,-65.483,-177.830,7.678,148.834
C08773=1143.580,226.256,-65.509,-177.827,7.681,148.834
C08774=1143.575,226.505,-65.534,-177.825,7.683,148.833
C08775=1143.570,226.753,-65.561,-177.822,7.686,148.833
C08776=1143.566,227.002,-65.587,-177.820,7.689,148.833
C08777=1143.562,227.251,-65.612,-177.816,7.692,148.833
C08778=1143.558,227.499,-65.638,-177.814,7.695,148.833
C08779=1143.552,227.747,-65.665,-177.811,7.698,148.833
C08780=1143.548,227.996,-65.691,-177.809,7.700,148.833
C08781=1143.544,228.245,-65.716,-177.806,7.703,148.833
C08782=1143.540,228.494,-65.742,-177.803,7.706,148.832
C08783=1143.535,228.742,-65.769,-177.800,7.708,148.832
C08784=1143.531,228.991,-65.795,-177.797,7.711,148.832
C08785=1143.526,229.239,-65.820,-177.794,7.714,148.832
C08786=1143.521,229.488,-65.847,-177.791,7.717,148.832
C08787=1143.517,229.736,-65.873,-177.789,7.719,148.832
C08788=1143.513,229.985,-65.899,-177.786,7.722,148.832
C08789=1143.508,230.234,-65.926,-177.784,7.725,148.832
C08790=1143.504,230.482,-65.952,-177.780,7.727,148.831
C08791=1143.500,230.731,-65.978,-177.778,7.730,148.831
C08792=1143.494,230.979,-66.004,-177.775,7.733,148.831
C08793=1143.490,231.228,-66.030,-177.772,7.736,148.831
C08794=1143.486,231.476,-66.057,-177.770,7.738,148.831
C08795=1143.481,231.725,-66.083,-177.767,7.741,148.831
C08796=1143.477,231.973,-66.109,-177.764,7.744,148.831
C08797=1143.473,232.222,-66.136,-177.761,7.747,148.831
C08798=1143.469,232.471,-66.162,-177.758,7.750,148.830
C08799=1143.464,232.720,-66.188,-177.755,7.753,148.830
C08800=1143.460,232.968,-66.215,-177.752,7.755,148.830
C08801=1143.455,233.217,-66.241,-177.750,7.758,148.830
C08802=1143.451,233.465,-66.268,-177.747,7.760,148.830
C08803=1143.447,233.714,-66.293,-177.745,7.763,148.830
C08804=1143.441,233.962,-66.320,-177.742,7.766,148.830
C08805=1143.437,234.210,-66.347,-177.739,7.769,148.830
C08806=1143.432,234.459,-66.373,-177.736,7.772,148.830
C08807=1143.429,234.707,-66.399,-177.733,7.775,148.829
C08808=1143.424,234.956,-66.426,-177.730,7.778,148.829
C08809=1143.419,235.229,-66.455,-177.727,7.781,148.829
C08810=1143.415,235.500,-66.484,-177.725,7.783,148.829
C08811=1143.409,235.772,-66.513,-177.721,7.787,148.829
C08812=1143.404,236.044,-66.542,-177.718,7.790,148.829
C08813=1143.400,236.292,-66.569,-177.716,7.793,148.829
C08814=1143.396,236.540,-66.596,-177.712,7.796,148.829
C08815=1143.391,236.789,-66.621,-177.710,7.799,148.829
C08816=1143.387,237.038,-66.649,-177.707,7.801,148.828
C08817=1143.382,237.286,-66.676,-177.705,7.804,148.828
C08818=1143.378,237.534,-66.702,-177.702,7.806,148.828
C08819=1143.373,237.784,-66.728,-177.699,7.809,148.828
C08820=1143.369,238.032,-66.755,-177.696,7.812,148.828
C08821=1143.365,238.281,-66.782,-177.693,7.815,148.828
C08822=1143.360,238.529,-66.809,-177.691,7.818,148.828
C08823=1143.357,238.778,-66.836,-177.688,7.821,148.828
C08824=1143.352,239.027,-66.862,-177.685,7.824,148.828
C08825=1143.347,239.275,-66.889,-177.682,7.827,148.828
C08826=1143.343,239.523,-66.916,-177.679,7.830,148.828
C08827=1143.338,239.772,-66.943,-177.677,7.833,148.828
C08828=1143.334,240.020,-66.970,-177.674,7.836,148.827
C08829=1143.330,240.269,-66.996,-177.671,7.839,148.827
C08830=1143.325,240.517,-67.023,-177.669,7.841,148.827
C08831=1143.320,240.766,-67.050,-177.666,7.844,148.827
C08832=1143.316,241.014,-67.077,-177.663,7.846,148.827
C08833=1143.312,241.262,-67.104,-177.660,7.849,148.827
C08834=1143.308,241.512,-67.131,-177.657,7.852,148.827
C08835=1143.303,241.760,-67.158,-177.654,7.855,148.827
C08836=1143.299,242.008,-67.185,-177.652,7.858,148.827
C08837=1143.295,242.257,-67.212,-177.649,7.861,148.827
C08838=1143.290,242.505,-67.239,-177.646,7.864,148.826
C08839=1143.285,242.754,-67.266,-177.643,7.867,148.826
C08840=1143.281,243.002,-67.293,-177.640,7.870,148.826
C08841=1143.277,243.251,-67.321,-177.638,7.872,148.826
C08842=1143.273,243.500,-67.347,-177.635,7.875,148.826
C08843=1143.268,243.748,-67.374,-177.632,7.878,148.826
C08844=1143.263,243.997,-67.401,-177.629,7.881,148.826
C08845=1143.259,244.245,-67.428,-177.627,7.884,148.826
C08846=1143.254,244.494,-67.455,-177.624,7.887,148.826
C08847=1143.251,244.742,-67.483,-177.621,7.890,148.826
C08848=1143.246,244.990,-67.510,-177.618,7.893,148.826
C08849=1143.242,245.239,-67.537,-177.615,7.896,148.826
C08850=1143.237,245.487,-67.564,-177.613,7.899,148.826
C08851=1143.232,245.736,-67.591,-177.610,7.902,148.825
C08852=1143.229,245.984,-67.619,-177.608,7.904,148.825
C08853=1143.224,246.233,-67.646,-177.605,7.907,148.825
C08854=1143.219,246.481,-67.673,-177.602,7.910,148.825
C08855=1143.215,246.730,-67.700,-177.599,7.913,148.825
C08856=1143.210,246.978,-67.728,-177.596,7.915,148.825
C08857=1143.206,247.227,-67.756,-177.594,7.918,148.825
C08858=1143.202,247.475,-67.783,-177.591,7.921,148.825
C08859=1143.198,247.723,-67.810,-177.588,7.924,148.825
C08860=1143.193,247.971,-67.837,-177.585,7.927,148.825
C08861=1143.189,248.221,-67.864,-177.582,7.930,148.825
C08862=1143.185,248.469,-67.892,-177.580,7.933,148.825
C08863=1143.180,248.717,-67.919,-177.577,7.936,148.825
C08864=1143.176,248.966,-67.947,-177.574,7.939,148.825
C08865=1143.172,249.214,-67.974,-177.572,7.942,148.825
C08866=1143.167,249.463,-68.001,-177.569,7.945,148.825
C08867=1143.162,249.711,-68.030,-177.566,7.948,148.824
C08868=1143.158,249.960,-68.057,-177.563,7.951,148.824
C08869=1143.154,250.208,-68.085,-177.561,7.954,148.824
C08870=1143.149,250.456,-68.112,-177.558,7.957,148.824
C08871=1143.145,250.706,-68.140,-177.555,7.960,148.824
C08872=1143.141,250.953,-68.167,-177.552,7.963,148.824
C08873=1143.136,251.201,-68.195,-177.549,7.965,148.824
C08874=1143.132,251.451,-68.222,-177.547,7.968,148.824
C08875=1143.128,251.698,-68.250,-177.544,7.971,148.824
C08876=1143.123,251.947,-68.277,-177.541,7.974,148.824
C08877=1143.120,252.195,-68.305,-177.538,7.977,148.824
C08878=1143.115,252.444,-68.333,-177.535,7.980,148.824
C08879=1143.110,252.692,-68.361,-177.533,7.983,148.824
C08880=1143.106,252.941,-68.388,-177.530,7.986,148.824
C08881=1143.101,253.189,-68.416,-177.528,7.989,148.824
C08882=1143.098,253.438,-68.444,-177.525,7.992,148.824
C08883=1143.093,253.686,-68.471,-177.522,7.995,148.824
C08884=1143.089,253.934,-68.499,-177.519,7.998,148.824
C08885=1143.084,254.183,-68.528,-177.516,8.001,148.823
C08886=1143.079,254.432,-68.555,-177.513,8.005,148.823
C08887=1143.075,254.679,-68.583,-177.510,8.008,148.823
C08888=1143.071,254.928,-68.611,-177.507,8.010,148.823
C08889=1143.067,255.176,-68.639,-177.505,8.013,148.823
C08890=1143.062,255.425,-68.667,-177.502,8.017,148.823
C08891=1143.058,255.673,-68.694,-177.499,8.020,148.823
C08892=1143.054,255.922,-68.723,-177.497,8.022,148.823
C08893=1143.050,256.170,-68.750,-177.494,8.025,148.823
C08894=1143.044,256.419,-68.778,-177.491,8.028,148.823
C08895=1143.041,256.667,-68.806,-177.488,8.031,148.823
C08896=1143.036,256.915,-68.834,-177.486,8.034,148.823
C08897=1143.032,257.164,-68.863,-177.483,8.037,148.823
C08898=1143.027,257.412,-68.890,-177.480,8.040,148.823
C08899=1143.024,257.660,-68.919,-177.478,8.043,148.823
C08900=1143.018,257.909,-68.946,-177.475,8.046,148.823
C08901=1143.015,258.158,-68.974,-177.472,8.049,148.823
C08902=1143.010,258.406,-69.002,-177.469,8.052,148.823
C08903=1143.006,258.654,-69.031,-177.466,8.055,148.823
C08904=1143.001,258.902,-69.059,-177.464,8.058,148.823
C08905=1142.998,259.151,-69.087,-177.461,8.061,148.823
C08906=1142.993,259.399,-69.115,-177.459,8.064,148.823
C08907=1142.989,259.648,-69.143,-177.456,8.067,148.823
C08908=1142.984,259.896,-69.172,-177.452,8.071,148.823
C08909=1142.980,260.144,-69.200,-177.450,8.074,148.823
C08910=1142.976,260.392,-69.228,-177.447,8.077,148.822
C08911=1142.971,260.641,-69.256,-177.444,8.080,148.822
C08912=1142.967,260.889,-69.284,-177.442,8.083,148.823
C08913=1142.962,261.163,-69.316,-177.439,8.086,148.823
C08914=1142.958,261.436,-69.347,-177.436,8.089,148.822
C08915=1142.953,261.709,-69.378,-177.433,8.092,148.822
C08916=1142.947,261.983,-69.409,-177.429,8.096,148.822
C08917=1142.944,262.232,-69.437,-177.427,8.099,148.822
C08918=1142.939,262.480,-69.466,-177.424,8.102,148.822
C08919=1142.935,262.728,-69.494,-177.421,8.105,148.822
C08920=1142.931,262.977,-69.523,-177.419,8.108,148.822
C08921=1142.926,263.225,-69.551,-177.416,8.111,148.822
C08922=1142.922,263.473,-69.580,-177.413,8.114,148.822
C08923=1142.918,263.721,-69.607,-177.410,8.117,148.822
C08924=1142.913,263.970,-69.636,-177.408,8.120,148.822
C08925=1142.909,264.219,-69.666,-177.405,8.124,148.822
C08926=1142.905,264.466,-69.693,-177.402,8.127,148.822
C08927=1142.900,264.715,-69.722,-177.399,8.130,148.822
C08928=1142.896,264.963,-69.750,-177.396,8.133,148.822
C08929=1142.891,265.211,-69.779,-177.394,8.136,148.822
C08930=1142.888,265.460,-69.808,-177.391,8.139,148.822
C08931=1142.883,265.708,-69.836,-177.388,8.142,148.822
C08932=1142.878,265.956,-69.865,-177.386,8.145,148.822
C08933=1142.875,266.205,-69.894,-177.383,8.148,148.822
C08934=1142.870,266.453,-69.922,-177.380,8.151,148.822
C08935=1142.865,266.701,-69.951,-177.377,8.155,148.822
C08936=1142.862,266.950,-69.979,-177.374,8.158,148.822
C08937=1142.857,267.198,-70.008,-177.371,8.161,148.822
C08938=1142.852,267.447,-70.037,-177.369,8.164,148.822
C08939=1142.849,267.695,-70.065,-177.366,8.167,148.822
C08940=1142.844,267.943,-70.095,-177.364,8.170,148.822
C08941=1142.839,268.192,-70.123,-177.361,8.173,148.822
C08942=1142.836,268.439,-70.152,-177.358,8.176,148.822
C08943=1142.831,268.688,-70.181,-177.356,8.179,148.822
C08944=1142.827,268.936,-70.210,-177.352,8.182,148.822
C08945=1142.822,269.185,-70.239,-177.349,8.185,148.822
C08946=1142.819,269.433,-70.268,-177.347,8.189,148.822
C08947=1142.814,269.681,-70.296,-177.344,8.192,148.822
C08948=1142.810,269.929,-70.325,-177.342,8.195,148.822
C08949=1142.805,270.178,-70.354,-177.339,8.197,148.822
C08950=1142.802,270.426,-70.383,-177.336,8.201,148.822
C08951=1142.796,270.674,-70.411,-177.333,8.204,148.822
C08952=1142.792,270.923,-70.441,-177.330,8.207,148.822
C08953=1142.788,271.171,-70.470,-177.328,8.211,148.822
C08954=1142.784,271.420,-70.499,-177.325,8.214,148.822
C08955=1142.780,271.667,-70.527,-177.322,8.217,148.822
C08956=1142.775,271.915,-70.557,-177.320,8.219,148.822
C08957=1142.771,272.164,-70.586,-177.317,8.223,148.822
C08958=1142.767,272.412,-70.615,-177.314,8.226,148.822
C08959=1142.763,272.661,-70.645,-177.311,8.229,148.822
C08960=1142.757,272.909,-70.673,-177.309,8.233,148.822
C08961=1142.753,273.157,-70.702,-177.306,8.236,148.822
C08962=1142.750,273.405,-70.731,-177.303,8.238,148.822
C08963=1142.746,273.653,-70.761,-177.301,8.242,148.822
C08964=1142.741,273.902,-70.789,-177.298,8.245,148.822
C08965=1142.737,274.150,-70.819,-177.295,8.248,148.822
C08966=1142.732,274.398,-70.848,-177.292,8.252,148.822
C08967=1142.728,274.646,-70.877,-177.290,8.255,148.822
C08968=1142.724,274.895,-70.907,-177.287,8.258,148.822
C08969=1142.719,275.143,-70.936,-177.284,8.260,148.822
C08970=1142.715,275.392,-70.965,-177.282,8.264,148.822
C08971=1142.711,275.640,-70.995,-177.278,8.267,148.822
C08972=1142.707,275.888,-71.024,-177.276,8.271,148.823
C08973=1142.703,276.137,-71.053,-177.273,8.274,148.823
C08974=1142.698,276.384,-71.083,-177.270,8.277,148.823
C08975=1142.694,276.632,-71.112,-177.268,8.280,148.823
C08976=1142.689,276.881,-71.141,-177.265,8.283,148.823
C08977=1142.685,277.129,-71.171,-177.262,8.287,148.823
C08978=1142.681,277.377,-71.200,-177.260,8.290,148.823
C08979=1142.677,277.625,-71.230,-177.257,8.293,148.823
C08980=1142.673,277.874,-71.259,-177.254,8.296,148.823
C08981=1142.669,278.122,-71.289,-177.252,8.299,148.823
C08982=1142.664,278.370,-71.318,-177.249,8.302,148.823
C08983=1142.660,278.619,-71.348,-177.246,8.306,148.823
C08984=1142.656,278.867,-71.377,-177.243,8.309,148.823
C08985=1142.652,279.115,-71.407,-177.240,8.312,148.823
C08986=1142.648,279.363,-71.436,-177.238,8.315,148.823
C08987=1142.643,279.611,-71.465,-177.235,8.318,148.823
C08988=1142.639,279.859,-71.495,-177.232,8.322,148.823
C08989=1142.635,280.107,-71.524,-177.230,8.325,148.823
C08990=1142.630,280.356,-71.554,-177.227,8.328,148.823
C08991=1142.626,280.604,-71.584,-177.224,8.331,148.823
C08992=1142.622,280.852,-71.614,-177.222,8.334,148.823
C08993=1142.617,281.100,-71.643,-177.218,8.338,148.823
C08994=1142.613,281.348,-71.673,-177.216,8.341,148.823
C08995=1142.609,281.597,-71.702,-177.213,8.344,148.823
C08996=1142.604,281.845,-71.732,-177.211,8.347,148.823
C08997=1142.600,282.093,-71.762,-177.208,8.350,148.823
C08998=1142.596,282.341,-71.792,-177.205,8.354,148.823
C08999=1142.592,282.589,-71.821,-177.202,8.357,148.824
C09000=1142.588,282.837,-71.851,-177.200,8.360,148.824
C09001=1142.583,283.086,-71.881,-177.197,8.363,148.824
C09002=1142.579,283.334,-71.911,-177.195,8.366,148.824
C09003=1142.575,283.582,-71.940,-177.192,8.370,148.824
C09004=1142.570,283.830,-71.971,-177.189,8.373,148.824
C09005=1142.566,284.079,-72.001,-177.186,8.377,148.824
C09006=1142.562,284.327,-72.030,-177.184,8.380,148.824
C09007=1142.558,284.575,-72.060,-177.180,8.383,148.824
C09008=1142.554,284.824,-72.091,-177.178,8.387,148.824
C09009=1142.550,285.071,-72.121,-177.175,8.389,148.824
C09010=1142.545,285.320,-72.150,-177.173,8.393,148.824
C09011=1142.541,285.568,-72.180,-177.170,8.396,148.824
C09012=1142.537,285.816,-72.210,-177.167,8.400,148.824
C09013=1142.532,286.064,-72.240,-177.164,8.403,148.824
C09014=1142.528,286.312,-72.271,-177.162,8.406,148.824
C09015=1142.524,286.560,-72.300,-177.159,8.409,148.824
C09016=1142.520,286.808,-72.330,-177.156,8.413,148.825
C09017=1142.515,287.084,-72.364,-177.154,8.416,148.825
C09018=1142.510,287.359,-72.397,-177.151,8.420,148.825
C09019=1142.506,287.635,-72.431,-177.147,8.424,148.825
C09020=1142.501,287.911,-72.464,-177.144,8.427,148.825
C09021=1142.497,288.159,-72.495,-177.142,8.431,148.825
C09022=1142.492,288.407,-72.525,-177.139,8.434,148.825
C09023=1142.488,288.655,-72.555,-177.136,8.437,148.825
C09024=1142.484,288.902,-72.585,-177.133,8.441,148.825
C09025=1142.480,289.151,-72.615,-177.131,8.444,148.825
C09026=1142.476,289.399,-72.645,-177.128,8.447,148.825
C09027=1142.472,289.647,-72.676,-177.126,8.450,148.825
C09028=1142.467,289.896,-72.706,-177.123,8.454,148.826
C09029=1142.463,290.144,-72.736,-177.120,8.457,148.826
C09030=1142.459,290.391,-72.767,-177.118,8.460,148.826
C09031=1142.454,290.639,-72.797,-177.115,8.463,148.826
C09032=1142.451,290.888,-72.827,-177.112,8.467,148.826
C09033=1142.446,291.136,-72.858,-177.109,8.470,148.826
C09034=1142.442,291.384,-72.888,-177.107,8.474,148.826
C09035=1142.438,291.632,-72.919,-177.104,8.477,148.826
C09036=1142.434,291.881,-72.949,-177.101,8.481,148.826
C09037=1142.429,292.129,-72.979,-177.098,8.484,148.826
C09038=1142.425,292.377,-73.010,-177.096,8.487,148.826
C09039=1142.421,292.624,-73.040,-177.094,8.490,148.826
C09040=1142.417,292.873,-73.072,-177.090,8.494,148.826
C09041=1142.413,293.121,-73.102,-177.088,8.497,148.827
C09042=1142.408,293.369,-73.132,-177.085,8.500,148.827
C09043=1142.404,293.617,-73.163,-177.082,8.504,148.827
C09044=1142.400,293.865,-73.193,-177.079,8.507,148.827
C09045=1142.396,294.113,-73.224,-177.077,8.510,148.827
C09046=1142.392,294.361,-73.254,-177.075,8.514,148.827
C09047=1142.387,294.609,-73.285,-177.071,8.517,148.827
C09048=1142.383,294.858,-73.316,-177.069,8.521,148.827
C09049=1142.379,295.105,-73.346,-177.066,8.523,148.827
C09050=1142.375,295.353,-73.377,-177.063,8.528,148.827
C09051=1142.371,295.602,-73.408,-177.061,8.531,148.828
C09052=1142.367,295.850,-73.438,-177.058,8.534,148.828
C09053=1142.362,296.098,-73.469,-177.055,8.538,148.828
C09054=1142.358,296.346,-73.500,-177.053,8.541,148.828
C09055=1142.354,296.594,-73.530,-177.050,8.544,148.828
C09056=1142.350,296.842,-73.561,-177.048,8.547,148.828
C09057=1142.346,297.090,-73.592,-177.045,8.551,148.828
C09058=1142.341,297.338,-73.623,-177.042,8.554,148.828
C09059=1142.337,297.585,-73.654,-177.040,8.558,148.828
C09060=1142.333,297.834,-73.685,-177.036,8.561,148.828
C09061=1142.329,298.082,-73.716,-177.034,8.565,148.829
C09062=1142.325,298.331,-73.747,-177.032,8.568,148.829
C09063=1142.320,298.579,-73.778,-177.028,8.572,148.829
C09064=1142.316,298.826,-73.808,-177.026,8.575,148.829
C09065=1142.313,299.074,-73.840,-177.023,8.578,148.829
C09066=1142.308,299.322,-73.870,-177.020,8.582,148.829
C09067=1142.303,299.570,-73.901,-177.018,8.585,148.829
C09068=1142.299,299.819,-73.932,-177.015,8.588,148.829
C09069=1142.295,300.066,-73.964,-177.012,8.592,148.829
C09070=1142.292,300.315,-73.994,-177.010,8.595,148.830
C09071=1142.287,300.563,-74.025,-177.008,8.599,148.830
C09072=1142.283,300.811,-74.056,-177.004,8.602,148.830
C09073=1142.279,301.059,-74.088,-177.002,8.606,148.830
C09074=1142.274,301.307,-74.118,-177.000,8.609,148.830
C09075=1142.270,301.555,-74.149,-176.996,8.613,148.830
C09076=1142.266,301.803,-74.181,-176.994,8.616,148.830
C09077=1142.262,302.051,-74.212,-176.992,8.619,148.831
C09078=1142.258,302.299,-74.244,-176.988,8.623,148.831
C09079=1142.254,302.547,-74.275,-176.986,8.626,148.831
C09080=1142.249,302.795,-74.305,-176.984,8.629,148.831
C09081=1142.245,303.043,-74.337,-176.981,8.634,148.831
C09082=1142.241,303.291,-74.368,-176.978,8.636,148.831
C09083=1142.236,303.538,-74.400,-176.976,8.640,148.831
C09084=1142.232,303.787,-74.431,-176.973,8.644,148.831
C09085=1142.228,304.034,-74.462,-176.970,8.647,148.831
C09086=1142.224,304.283,-74.493,-176.968,8.650,148.832
C09087=1142.220,304.530,-74.525,-176.965,8.654,148.832
C09088=1142.216,304.779,-74.556,-176.962,8.657,148.832
C09089=1142.211,305.026,-74.587,-176.960,8.660,148.832
C09090=1142.207,305.275,-74.618,-176.957,8.664,148.832
C09091=1142.204,305.523,-74.650,-176.954,8.668,148.832
C09092=1142.199,305.771,-74.682,-176.951,8.672,148.833
C09093=1142.195,306.019,-74.713,-176.949,8.675,148.833
C09094=1142.191,306.267,-74.744,-176.946,8.678,148.833
C09095=1142.187,306.515,-74.776,-176.943,8.682,148.833
C09096=1142.183,306.763,-74.807,-176.941,8.685,148.833
C09097=1142.179,307.011,-74.839,-176.939,8.688,148.833
C09098=1142.174,307.259,-74.870,-176.935,8.692,148.833
C09099=1142.170,307.507,-74.902,-176.933,8.696,148.834
C09100=1142.166,307.754,-74.934,-176.930,8.700,148.834
C09101=1142.162,308.003,-74.965,-176.928,8.703,148.834
C09102=1142.158,308.251,-74.997,-176.925,8.706,148.834
C09103=1142.154,308.498,-75.028,-176.922,8.710,148.834
C09104=1142.150,308.746,-75.060,-176.920,8.713,148.834
C09105=1142.145,308.994,-75.092,-176.917,8.716,148.834
C09106=1142.141,309.243,-75.123,-176.914,8.720,148.835
C09107=1142.137,309.491,-75.155,-176.912,8.724,148.835
C09108=1142.133,309.738,-75.186,-176.909,8.727,148.835
C09109=1142.129,309.986,-75.218,-176.906,8.731,148.835
C09110=1142.125,310.234,-75.251,-176.904,8.734,148.835
C09111=1142.120,310.482,-75.282,-176.901,8.738,148.835
C09112=1142.116,310.730,-75.313,-176.899,8.741,148.836
C09113=1142.113,310.978,-75.345,-176.896,8.745,148.836
C09114=1142.108,311.226,-75.377,-176.893,8.749,148.836
C09115=1142.104,311.474,-75.409,-176.891,8.752,148.836
C09116=1142.100,311.722,-75.441,-176.888,8.756,148.836
C09117=1142.095,311.970,-75.473,-176.885,8.759,148.836
C09118=1142.092,312.218,-75.505,-176.883,8.763,148.837
C09119=1142.088,312.466,-75.537,-176.880,8.766,148.837
C09120=1142.083,312.713,-75.568,-176.878,8.770,148.837
C09121=1142.078,312.991,-75.604,-176.875,8.774,148.837
C09122=1142.074,313.269,-75.640,-176.872,8.777,148.837
C09123=1142.070,313.547,-75.677,-176.869,8.781,148.837
C09124=1142.065,313.825,-75.711,-176.866,8.786,148.838
C09125=1142.060,314.072,-75.744,-176.863,8.790,148.838
C09126=1142.057,314.320,-75.776,-176.860,8.793,148.838
C09127=1142.053,314.568,-75.808,-176.858,8.797,148.838
C09128=1142.048,314.817,-75.840,-176.855,8.800,148.839
C09129=1142.044,315.064,-75.872,-176.853,8.803,148.839
C09130=1142.040,315.312,-75.904,-176.850,8.808,148.839
C09131=1142.036,315.560,-75.936,-176.848,8.811,148.839
C09132=1142.033,315.808,-75.969,-176.844,8.815,148.839
C09133=1142.028,316.055,-76.001,-176.842,8.818,148.839
C09134=1142.024,316.304,-76.033,-176.839,8.822,148.840
C09135=1142.019,316.552,-76.065,-176.837,8.825,148.840
C09136=1142.016,316.800,-76.097,-176.834,8.828,148.840
C09137=1142.012,317.048,-76.130,-176.831,8.832,148.840
C09138=1142.007,317.295,-76.162,-176.829,8.836,148.840
C09139=1142.003,317.543,-76.194,-176.826,8.840,148.841
C09140=1141.999,317.791,-76.226,-176.824,8.843,148.841
C09141=1141.995,318.039,-76.259,-176.821,8.847,148.841
C09142=1141.991,318.287,-76.291,-176.819,8.850,148.841
C09143=1141.986,318.535,-76.323,-176.816,8.854,148.841
C09144=1141.983,318.782,-76.355,-176.813,8.858,148.842
C09145=1141.978,319.031,-76.388,-176.810,8.862,148.842
C09146=1141.975,319.278,-76.420,-176.808,8.865,148.842
